# B&R Automation Studio project ABC_Pltzr (part 2)

### bgringbuffer.c
```c
#ifndef _BG_RINGBUFFER_C
#define _BG_RINGBUFFER_C
/*
File:
bgRingBuffer.c

About:
------
- ring buffer implementation

B&R System Dependencies:
------------------------
- B&R system library: none
- B&R system header files: stdarg.h

History:
--------
03/11/2005
-first version

Test and example code:
----------------------
- to run this file standalone:
--- enable following code section (remove or comment out #if 0 / #endif)
--- create cyclic object (task) from C Language and add this file
*/
#include <stdarg.h>

#include <bur/plctypes.h>
#ifdef _DEFAULT_INCLUDES
	#include <AsDefault.h>
#endif

#include "bgringbuffer.h"
//#include "bgdebug.h"

//#include "bgsprintf.h"
//#include "bgsprintf.c"

#if 0
#include<bur/plc.h>
#include <bur/plctypes.h>

//#include <bgsprintf.h>
#include <bgringbuffer.h>

_LOCAL int counter;

_LOCAL bgRingBuffer_typ myRB;

#define TXT_SIZE 64
_LOCAL char textBuffer1[TXT_SIZE];
_LOCAL char textBuffer2[TXT_SIZE];

#define RB_SIZE 64
_LOCAL char ringBuffer[RB_SIZE];

_INIT void Init(void) {

	rbInit(&myRB, ringBuffer, RB_SIZE);
}

_CYCLIC void Cyclic(void) {

	counter++;

	sprintf2(textBuffer1, "Counter=%d\n", counter);
	bgRingBuffPutString(&myRB, textBuffer1);
    bgRingBuffGet(&myRB, textBuffer2, TXT_SIZE);
}
#endif
/*End: Example/Test code*/

static char *bgRingBuffGetPtrToFileName(char *pFileNameWithPath)
{
/*
Input Example:
*pFileNameWithPath = "d:/data/temp/cobble/2005-9-1/new_ng.pgp/pgm/new_ng/cpu/bgstatemachine.c"
                                                                             |
Output value is ptr to: bgstatemachine.c ------------------------------------+
*/
int i;
int len = brsstrlen((UDINT)pFileNameWithPath);
char* pStart = (char*)(pFileNameWithPath + len);
	for(i=0;i<len; i++, pStart--){
		if( (*pStart == '/') || (*pStart == '\\') ){
			pStart++;
			return pStart;
		}
	}
	return pFileNameWithPath;
}

static void bgRingBuffIncDataInPtr(bgRingBuffer_typ *rb){
	rb->ptrDataIn++;
    if(rb->ptrDataIn >= rb->ptrCircularBufferEnd){
    	rb->ptrDataIn = rb->ptrCircularBufferBegin;
#if 0
/*mark wrap arround for testing*/
    	*rb->ptrDataIn = '@';
    	rb->ptrDataIn++;
#endif
    }
}

static void bgRingBuffIncDataOutPtr(bgRingBuffer_typ *rb){
	rb->ptrDataOut++;
	if(rb->ptrDataOut >= rb->ptrCircularBufferEnd)
		rb->ptrDataOut = rb->ptrCircularBufferBegin;
}

void bgRingBuffInit(bgRingBuffer_typ *rb, char *buffer, int bufSize)
{
	if(!buffer || !bufSize)
		return;

	rb->init = 1;
	rb->overrun = 0;
	rb->bufSize = bufSize;
    rb->ptrCircularBufferBegin = buffer;
    rb->ptrCircularBufferEnd = buffer + rb->bufSize;
    rb->ptrDataIn = rb->ptrCircularBufferBegin;
    rb->ptrDataOut = rb->ptrCircularBufferBegin;
}
/*
----------------------------------------------------------
*/
void bgRingBuffPutString(bgRingBuffer_typ *rb, char *sourceString)
{
    char *src = sourceString;

	if(!rb->init)
		return;

    /*input is string! look for zero termination*/
    while( *src ){

        /*store char*/
        *rb->ptrDataIn = *src;

        /*inc ptrs*/
		src++;

        bgRingBuffIncDataInPtr(rb);

        /*check if ring-buffer full*/
        if(rb->ptrDataIn == rb->ptrDataOut){
        	/*move out ptr one step ahead of in ptr*/
	        bgRingBuffIncDataOutPtr(rb);

			/*mark ring buffer overrun*/
			if(!rb->overrun){
		        char text[3]={'<','?','>'};
		        int i;
				rb->overrun = 1;
	        	for(i=0;i<3;i++){
			        *rb->ptrDataIn = text[i];
			        bgRingBuffIncDataInPtr(rb);
			        bgRingBuffIncDataOutPtr(rb);
		        }
		    }
        }
    }
}
/*
----------------------------------------------------------
*/
int bgRingBuffGet(bgRingBuffer_typ *rb, char *destination, int destSize)
{
char *dst = destination;
char *dstMax = dst + destSize;
int length = 0;

	if(!rb->init)
		return 0;

    if(rb->ptrDataIn == rb->ptrDataOut)
        return 0;

    while(1){
        *dst = *rb->ptrDataOut;
		length++;

        dst++;
        /*check if max size riched*/
        if(dst >= dstMax)
            break;

  		bgRingBuffIncDataOutPtr(rb);

        /*check if ring-buffer empty*/
        if(rb->ptrDataIn == rb->ptrDataOut){

        	/*mark end of ring buffer overrun*/
			if(rb->overrun){
		        char text[3]={'<','!','>'};
		        int i;

				rb->overrun = 0;
	        	for(i=0;i<3;i++){
			        *dst = text[i];
			        dst++;
			        length++;
			        if(dst >= dstMax)
			            break;
		        }
		    }

            break;
        }
    }
    return length;
}

void bgRingBuffPutDbgInfo(bgRingBuffer_typ *rb, char *file, char *function, unsigned int level, unsigned int unused, char *format, ...)
{
char txt[256];

va_list args;

	/*if dbg entry level > then currently set dbg level -> exit*/
	if( level > rb->dbgLevel )
		return;

	/*timestap needed? default=no*/
	if( rb->dbgFormat & BG_DEBUG_FORMAT_LEVEL){
		switch(level){
			case 0: bgRingBuffPutString(rb, "CRT|"); break;
			case 1: bgRingBuffPutString(rb, "ERR|"); break;
			case 2: bgRingBuffPutString(rb, "WAR|"); break;
			case 3: bgRingBuffPutString(rb, "INF|"); break;
			case 4: bgRingBuffPutString(rb, "DBG|"); break;
			default: bgRingBuffPutString(rb, "???|"); break;
		}
	}

	/*timestap needed? default=no*/
	if( rb->dbgFormat & BG_DEBUG_FORMAT_TIMESTAMP){
//		bgsprintf(txt, "%s|", "2005-10-01 12:32:44.123" );
//		bgRingBuffPutString(rb, txt);
	}

	/*filename needed? default=no*/
	if( rb->dbgFormat & BG_DEBUG_FORMAT_FILENAME){
//		bgsprintf(txt, "%s|", bgRingBuffGetPtrToFileName(file) );
//		bgRingBuffPutString(rb, txt);
	}

	/*function name needed? default=no*/
	if( rb->dbgFormat & BG_DEBUG_FORMAT_FUNCTION){
//		bgsprintf(txt, "%s()|", function);
//		bgRingBuffPutString(rb, txt);
	}

    va_start( args, format );

//	bgvsprintf(txt, format, args);
//	bgvsprintf(txt, format, args);

	bgRingBuffPutString(rb, txt);
}

#if 0
void bgRingBuffPrintf(bgRingBuffer_typ *rb, char *format, ...)
{
char txt[256];
va_list ap;
int num;

    va_start( ap, format );

//	bgvsprintf(txt, format, args);

	num = __ofmt(0, txt, 256, format, ap);

	va_end(ap);
//	return num;

	bgRingBuffPutString(rb, txt);
}
#endif

#endif
/*EOF*/
```

### bgsscanf.h
```c
/*
File:
bgsscanf.h

About:
------
- short and limited implementation of the sscanf() function

*/
#ifndef _BG_SSCANF_H
#define _BG_SSCANF_H

#include <stdarg.h>

/*
Public data types:
-----------------
*/

/*
Public functions:
-----------------
*/
int bgsscanf(const char *out, const char *format, ...);

int bgvsscanf(const char *out, const char *format, va_list args);

#endif
```

### bgstring.c
```c
#ifndef _BG_STRING_C
#define _BG_STRING_C

#ifdef WIN32
#include "string.h"
#else
#include <bur/plctypes.h>
#endif
#include "bgstring.h"

/*
File:
bgString.c

About:
------
- implements  additional string manipulation functions

B&R System Dependencies:
------------------------
- B&R system library: libasstring.a
- B&R system header files: asstring.h

History:
--------
09/11/2005
- rectified issue with bgStringListLines() to properly handle zero length
input string

05/08/2005
-first version

Test and example code:
----------------------
- to run this file standalone:
--- enable following code section (remove or comment out #if 0 / #endif)
--- create cyclic object (task) from C Language and add this file
*/

#if 0
#include <bur/plc.h>
#include <bur/plctypes.h>

#define TXT_SIZE 64
_LOCAL char textBuffer1[TXT_SIZE];
_LOCAL char textBuffer2[TXT_SIZE];
_LOCAL int idxResult;
_LOCAL int idxStart;
_LOCAL int idxEnd;

_INIT void Init(void) {

	/*use defaults*/
	idxStart 	= -1;
	idxEnd 		= -1;
	/*start with empty strings*/
	textBuffer1[0] = 0;
	textBuffer2[0] = 0;
}

_CYCLIC void Cyclic(void) {

	idxResult = bgStrFind(textBuffer1, textBuffer2, start, end);

}
#endif

/*End: Example/Test code*/
int bgStrFind(char *s, char *sub, int idxStart, int idxEnd)
{
	int i, j;
	int subLen;
	char *ptrStr;
	char *ptrSub;

	/*exit if null ptrs*/
	if(!s || !sub)
		return -1;

	/*exit if zero strings*/
	if( !(*s) || !(*sub) )
		return -1;

	subLen = brsstrlen((UDINT)sub);

	/*check starting index: default = -1 -> start @ s[0]*/
	if(idxStart < 0)
		idxStart = 0;

	/*check end index: default = -1 -> end is sLength - subLength*/
	if(idxEnd < 0){
		idxEnd = brsstrlen((UDINT)s) - subLen;
	}

	/*check if start is beyond the end*/
	if(idxStart > idxEnd)
		return -1;

	/*search for string <sub> within the string <s>*/
	for(i=idxStart; i<=idxEnd; i++)
	{
		ptrStr = s + i;
		ptrSub = sub;

		for(j=0; j<subLen; j++, ptrStr++, ptrSub++)
		{
			if( *ptrStr!= *ptrSub)
				break;
		}

		if( j == subLen)
			return i;
	}

	return -1;
}

/*
bgStrFindEx - has an extra option
option = 0; same as bgStrFind
option = 1; before comparing, both strings are converted to lower case
*/
int bgStrFindEx(char *s, char *sub, int idxStart, int idxEnd, int option)
{
	int i, j;
	int subLen;
	char *ptrStr;
	char *ptrSub;

	/*exit if null ptrs*/
	if(!s || !sub)
		return -1;

	/*exit if zero strings*/
	if( !(*s) || !(*sub) )
		return -1;

	subLen = brsstrlen((UDINT)sub);

	/*check starting index: default = -1 -> start @ s[0]*/
	if(idxStart < 0)
		idxStart = 0;

	/*check end index: default = -1 -> end is sLength - subLength*/
	if(idxEnd < 0){
		idxEnd = brsstrlen((UDINT)s) - subLen;
	}

	/*check if start is beyond the end*/
	if(idxStart > idxEnd)
		return -1;

	/*search for string <sub> within the string <s>*/
	for(i=idxStart; i<=idxEnd; i++)
	{
		ptrStr = s + i;
		ptrSub = sub;

		for(j=0; j<subLen; j++, ptrStr++, ptrSub++)
		{
			if(!option){
				if( *ptrStr!= *ptrSub)
					break;
			}else{
				if( bgCharToLowerCase(*ptrStr) != bgCharToLowerCase(*ptrSub) )
					break;
			}
		}

		if( j == subLen)
			return i;
	}

	return -1;
}

int bgStrCpyN(char *dest, char *src, int maxNoOfCharsToCopy)
{
int i;

	/*maxNoOfCharsToCopy-1 - takes into consideration that supplied max
	length is usually the buffer size, 1 char is needed for null termination
	*/
	for(i=0; i<(maxNoOfCharsToCopy-1);i++){
		*(dest+i)=*(src+i);
		if(! (*(src+i) ) )
			break;
	}

	/*if max reached, terminate dest string*/
	if(i >= (maxNoOfCharsToCopy-1))
		*(dest+i)=0;

	/*string termination is not included in the string length*/
	return i;
}

int bgStrTrimCRLF(char *s)
{
int i;
char c;

	for(i=0;i<255;i++){

		c = s[i];

		if( !c )
			break;

		if( (c == 0xa) || (c == 0xd) ){
			s[i] = 0;
			break;
		}
	}

	return i;
}

int bgStrCpyNTrimLeadingSpaces(char *dest, char *src, int maxNoOfCharsToCopy)
{
int i;
int found;
char *srcStart;

	/*look for leading spaces*/
	found = 0;
	for(i=0; i<(maxNoOfCharsToCopy-1);i++){
		if( *(src+i) != ' ' ){
			srcStart = src + i;
			found = 1;
			break;
		}
	}

	if(!found){
	/*src string is all spaces->set destination to empty string*/
		*dest = 0;
		return 0;
	}

	return bgStrCpyN(dest, srcStart, maxNoOfCharsToCopy);
}

/*
copy string, don't go over the size of dest buffer, trim leading / trailing spaces / convert
to lower case
*/
int bgStrCpyNTrimSpcsToLwr(char *dest, char *src, int maxNoOfCharsToCopy)
{
int i;
char* srcStart = src;
char* srcEnd;
int len = brsstrlen((UDINT)src);

	if( !len )
		return len;

	/*find src start, avoid leading spaces*/
	while(1){
		if( *srcStart != ' ')
			break;

		if( *srcStart == 0)
			return 0;

		srcStart++;
	}

	/*find src end, trim trailing spaces*/
	srcEnd = (char*)(src + len - 1);
	while(1){
		if( *srcEnd != ' ')
			break;

		if( *srcEnd == 0)
			return 0;

		srcEnd--;
	}

	srcEnd++;

	if( srcStart >= srcEnd )
		return 0;

	for(i=0; i<(maxNoOfCharsToCopy-1); i++){
		dest[i] = bgCharToLowerCase(*srcStart);
		srcStart++;
		if(srcStart >= srcEnd){
			i++;
			break;
		}
	}

	dest[i] = 0;
	return i;
}

int bgIsDigit(char c){
	return ((c>='0') && (c<='9')) ? 1 : 0;
}

#if 0
/*
Test for: bgStringListLinesEx()

The xxxxEx functions use externaly supplied buffer space to store result pointers to
lines / words.
Based on the supplied buffer size, functions will calculate max. number of items (char ptr-s)
that may be stored within the given / allocated storage area.
See: pList->itemCountMax

To test it out, create a new cyclic task then use following code!
*/
#include <bur/plc.h>
#include <bur/plctypes.h>

#include "bglib/bgString.h"
#include "bglib/bgString.c"

#include "bglib/bgdebug.h"
#include "bglib/bgringbuffer.c"

_LOCAL bgStringListEx_typ listLines;
_LOCAL bgStringListEx_typ listWords;
_LOCAL char multiLineTextBuffer[256];
_LOCAL int lineCount;
_LOCAL int wordCount;
_LOCAL int test;
_LOCAL char listPtrBuf[128];    /*this is a "free" storage for list ptr-s! use it with caution!*/

_INIT void init()
{
	strcpy(multiLineTextBuffer, "hello world\r\nThis is a test for second line!\r\nThird line is here and there...\r\nLine #4 : right.left dot !\r\n");
	test = 0;
}

_CYCLIC void cyclic()
{
int i, j;

/*
This is just an example on how to use external / user supplied buffer in order to
store line / word lists. Based on the supplied buffer size, functions will calculate
max. number of items that may be stored within the given / allocated storage area.
See: pList->itemCountMax
*/
char* lineListStorage = &listPtrBuf[0];
char* wordListStorage = &listPtrBuf[64];

	if( test ){
		test = 0;

		lineCount = bgStringListLinesEx(&listLines, multiLineTextBuffer, lineListStorage, 64);
		DBG("multiLineTextBuffer has lineCount=%d lines. (same as listLines.itemCount= %d). Lines are:\r\n", lineCount, listLines.itemCount);
		for(i=0; i<listLines.itemCount; i++){
			DBG("Line[%d]->%s\r\n", i, listLines.items[i]);
			wordCount = bgStringSplitLineEx(&listWords, ' ', listLines.items[i], wordListStorage, 64);
				DBG("     Line[%d] has wordCount=%d words. (same as listWords.itemCount= %d). Words are:\r\n", i, wordCount, listWords.itemCount)
			for(j = 0; j<listWords.itemCount; j++)
				DBG("     Word[%d]->%s\r\n", j, listWords.items[j]);
		}
	}
}
#endif
int bgStringListLines(bgStringList_typ * p){
unsigned char *ptrItemStart, *ptrItemEnd;
int	calcItemCount;

/*
	length = strlen( p->src );
*/
	p->itemCount = 0;

	ptrItemStart = p->src;
	ptrItemEnd = p->src;

	if( *ptrItemStart == 0){
		return 0;
	}

/*process the rest; build list of item pointers*/
	calcItemCount 	= 0;
	while( 1 ){
		if( (*ptrItemEnd == 0x0D) || (*ptrItemEnd == 0x0A)){
			*ptrItemEnd = 0;
			p->items[calcItemCount] = ptrItemStart;
			ptrItemEnd++;

			/*check for an additional \r or \n*/
			if( (*ptrItemEnd == 0x0D) || (*ptrItemEnd == 0x0A)){
				ptrItemEnd++;
			}

			ptrItemStart = ptrItemEnd;
			calcItemCount++;

			if(calcItemCount >= BG_STRINGLIST_MAXITEMCOUNT){
				p->itemCount = calcItemCount;
				return -1;
			}

			/*check for an end of the src string*/
			if( (*ptrItemEnd == 0) ){
				p->itemCount = calcItemCount;
				return calcItemCount;
			}
		}else
		if( *ptrItemEnd == 0){
			p->items[calcItemCount] = ptrItemStart;
			calcItemCount++;
			break;
		}else
			ptrItemEnd++;
	}/*while*/

	p->itemCount = calcItemCount;
	return calcItemCount;
}

void bgStringListExMemSet(bgStringListEx_typ *p, char* pAddrListBuffer, int sizeListBuffer)
{
	/*NOTE: we are going to use supplied char buffer as the storage for the array of char ptr-s!*/
    p->items = (unsigned char**)pAddrListBuffer;

	p->itemCountMax = sizeListBuffer / sizeof(char*);
}

int bgStringListLinesEx(bgStringListEx_typ * p, char* pContentBuffer, char* pAddrListBuffer, int sizeListBuffer){
unsigned char *ptrItemStart, *ptrItemEnd;
int	calcItemCount;

    p->src = (unsigned char*)pContentBuffer;

    /*if mem data is defined, use it; otherwise, mem shall have been set using a separate call to xxxExMemSet()*/
    if(pAddrListBuffer && sizeListBuffer)
        bgStringListExMemSet(p, pAddrListBuffer, sizeListBuffer);

	p->itemCount = 0;

	ptrItemStart = p->src;
	ptrItemEnd = p->src;

	if( *ptrItemStart == 0){
		return 0;
	}

/*process the rest; build list of item pointers*/
	calcItemCount 	= 0;
	while( 1 ){
		if( (*ptrItemEnd == 0x0D) || (*ptrItemEnd == 0x0A)){
			*ptrItemEnd = 0;
			p->items[calcItemCount] = ptrItemStart;
			ptrItemEnd++;

			/*check for an additional \r or \n*/
			if( (*ptrItemEnd == 0x0D) || (*ptrItemEnd == 0x0A)){
				ptrItemEnd++;
			}

			ptrItemStart = ptrItemEnd;
			calcItemCount++;

			if(calcItemCount >= p->itemCountMax){
				p->itemCount = calcItemCount;
				return -1;
			}

			/*check for an end of the src string*/
			if( (*ptrItemEnd == 0) ){
				p->itemCount = calcItemCount;
				return calcItemCount;
			}
		}else
		if( *ptrItemEnd == 0){
			p->items[calcItemCount] = ptrItemStart;
			calcItemCount++;
			break;
		}else
			ptrItemEnd++;
	}/*while*/

	p->itemCount = calcItemCount;
	return calcItemCount;
}

#if 0
Example:
(AS: Make a "C" task; add <filename>.c to the task; copy & paste this code)
#######
#include <bur/plc.h>
#include <bur/plctypes.h>

#include "bgString.h"
#include "bgString.c"

#include "bgdebug.h"

_LOCAL bgStringList_typ myList;
_LOCAL bgStringList_typ mySplitList;
_LOCAL char buffer[256];
_LOCAL int lineCount;
_LOCAL int test;

_INIT void init()
{
	strcpy(buffer, "hello world\r\nwhat is new?\r\nthird line\r\nline #4\r\n");
	test = 0;
}

_CYCLIC void cyclic()
{
int i, j;

	if( test ){
		test = 0;
		myList.src = buffer;
		lineCount = bgStringListLines(&myList);

		for(i=0; i<myList.itemCount; i++){
			DBG("Line[%d]->%s\r\n", i, myList.items[i]);

			mySplitList.src = myList.items[i];
			lineCount = bgStringSplitLine(&mySplitList, ' ');
			for(j = 0; j<mySplitList.itemCount; j++)
				DBG("     Word[%d]->%s\r\n", j, mySplitList.items[j]);
		}
	}
}
######
The above code generates following output (debug telnet client):
>Line[0]->hello world
     Word[0]->hello
     Word[1]->world
Line[1]->what is new?
     Word[0]->what
     Word[1]->is
     Word[2]->new?
Line[2]->third line
     Word[0]->third
     Word[1]->line
Line[3]->line #4
     Word[0]->line
     Word[1]->#4

#endif
int bgStringSplitLine(bgStringList_typ * p, char separator){
unsigned char *ptrItemStart, *ptrItemEnd;
int	calcItemCount;

	p->itemCount = 0;

	ptrItemStart = p->src;
	ptrItemEnd = p->src;

/*process the rest; build list of item pointers*/
	calcItemCount 	= 0;
	while( 1 ){
		if( (*ptrItemEnd == separator) ){
			*ptrItemEnd = 0;
			p->items[calcItemCount] = ptrItemStart;
			ptrItemEnd++;

			calcItemCount++;

			/*check for an additional separtor */
			while( (*ptrItemEnd == separator) ){
				ptrItemEnd++;
				if( (*ptrItemEnd == 0) ){
					p->itemCount = calcItemCount;
					return calcItemCount;
				}
			}

			ptrItemStart = ptrItemEnd;

			if(calcItemCount >= BG_STRINGLIST_MAXITEMCOUNT){
				p->itemCount = calcItemCount;
				return -1;
			}

			/*check for an end of the src string*/
			if( (*ptrItemEnd == 0) ){
				p->itemCount = calcItemCount;
				return calcItemCount;
			}
		}else
		if( *ptrItemEnd == 0){
			p->items[calcItemCount] = ptrItemStart;
			calcItemCount++;
			break;
		}else
			ptrItemEnd++;
	}/*while*/

	p->itemCount = calcItemCount;
	return calcItemCount;
}

int bgStringSplitLineEx(bgStringListEx_typ * p, char separator, char* pLineBuffer, char* pAddrListBuffer, int sizeListBuffer){
unsigned char *ptrItemStart, *ptrItemEnd;
int	calcItemCount;

    p->src = (unsigned char*)pLineBuffer;

    /*if mem data is defined, use it; otherwise, mem shall have been set using a separate call to xxxExMemSet()*/
    if(pAddrListBuffer && sizeListBuffer)
        bgStringListExMemSet(p, pAddrListBuffer, sizeListBuffer);

	p->itemCount = 0;

	ptrItemStart = p->src;
	ptrItemEnd = p->src;

/*process the rest; build list of item pointers*/
	calcItemCount 	= 0;
	while( 1 ){
		if( (*ptrItemEnd == separator) ){
			*ptrItemEnd = 0;
			p->items[calcItemCount] = ptrItemStart;
			ptrItemEnd++;

			calcItemCount++;

			/*check for an additional separtor */
			while( (*ptrItemEnd == separator) ){
				ptrItemEnd++;
				if( (*ptrItemEnd == 0) ){
					p->itemCount = calcItemCount;
					return calcItemCount;
				}
			}

			ptrItemStart = ptrItemEnd;

			if(calcItemCount >= p->itemCountMax){
				p->itemCount = calcItemCount;
				return -1;
			}

			/*check for an end of the src string*/
			if( (*ptrItemEnd == 0) ){
				p->itemCount = calcItemCount;
				return calcItemCount;
			}
		}else
		if( *ptrItemEnd == 0){
			p->items[calcItemCount] = ptrItemStart;
			calcItemCount++;
			break;
		}else
			ptrItemEnd++;
	}/*while*/

	p->itemCount = calcItemCount;
	return calcItemCount;
}

char *bgStringLower(char *s)
{
int i;
char c;

	for(i=0;i<255;i++){

		c = s[i];

		if( !c )
			break;

		if( (c >= 'A') && (c <= 'Z') ){
			s[i] = c - 'A' + 'a';
		}
	}

	return s;
}

char bgCharToLowerCase(char c)
{
char charLowerCase = c;

	if( (c >= 'A') && (c <= 'Z') ){
		charLowerCase = c - 'A' + 'a';
	}

	return charLowerCase;
}

char *bgStringUpper(char *s)
{
int i;
char c;

	for(i=0;i<255;i++){

		c = s[i];

		if( !c )
			break;

		if( (c >= 'a') && (c <= 'z') ){
			s[i] = c - 'a' + 'A';
		}
	}

	return s;
}

int bgStringIsMatch(char *s1, char *s2, int minChrCount)
{
	if( !brsstrcmp((UDINT)s1, (UDINT)s2) ){
		return 1;
	}else
		return 0;

}

int bgIsNumber_uint(char *s)
{
int i;
char c;

	/*limit execution to 255: don't want cycle time violation due to wrong ptr*/
	for(i=0;i<255;i++){

		c = s[i];

		/*end of valid input string?*/
		if( !c && i)
			return 1;

		/*zero input string?*/
		if( !c && !i)
			return 0;

		/*check if digit or space*/
		if( !bgIsDigit(c) && (c != ' '))
			return 0;
	}

	return 0;
}

int bgIsNumber_int(char *s)
{
int i;
char c;

	/*limit execution to 255: don't want cycle time violation due to wrong ptr*/
	for(i=0;i<255;i++){

		c = s[i];

		/*end of valid input string?*/
		if( !c && i)
			return 1;

		/*zero input string?*/
		if( !c && !i)
			return 0;

		/*check if digit or space*/
		if( !bgIsDigit(c) && (c != ' ') && (c != '-')  && (c != '+'))
			return 0;
	}

	return 0;
}

int bgAsciiToUint(char *src, unsigned int *dst)
{

unsigned int value;

	if( !bgIsNumber_uint(src) )
		return 0;

#ifdef WIN32
	/*TODO!!!*/
	value = 0;
#else
	value = brsatoi((UDINT)src);
#endif

	*dst = value;

	return 1;
}

int bgAsciiToInt(char *src, unsigned int *dst)
{

unsigned int value;

	if( !bgIsNumber_int(src) )
		return 0;

#ifdef WIN32
	/*TODO!!!*/
	value = 0;
#else
	value = brsatoi((UDINT)src);
#endif
	*dst = value;

	return 1;
}

int bgStrCopyFromTo(char* src, int srcStartPosition, int srcEndPosition, char* dest)
{
/*
-copy part of the memory from the section of src (from srcStartPosition to srcEndPosition) to dest
-srcEndPosition is not included in the copy (last copied byte position is srcEndPosition-1)
-length of the copied string is (srcEndPosition - srcStartPosition)
Example:
src="01234567890"
srcStartPosition=3
srcEndPosition=7

dest="3456"

return value: number of bytes copied (i.e. length of the dest string)
*/
int size = 0;
int i;

	if( srcEndPosition >= srcStartPosition )
		size = srcEndPosition - srcStartPosition;

	/*do memcopy! end position char is not included in the copy!*/
	for(i=0; i<size; i++)
		dest[i] = src[srcStartPosition + i];

	/*terminate string*/
	dest[size] = 0;

	return size;
}

int bgStrFindEOL(char* src, int startPosition)
{
/*
- search supplied c string "src" (zero terminated!!!) for the eof
- start search at startPosition and look for the first '\n'
- return:
-1 		- EOF (\n) not found
>=0		- EOF position
*/
int position = startPosition;
int i = 0;

	while(1){
		/*end of line?*/
		if( src[position] == '\n' ){
			/*if \r preceeds \n, dec EOL position by 1*/
			if( position && (src[position-1] == '\r') )
				position--;

		 	return position;
		}

 		/*end of string?*/
		if( src[position] == 0 ) return -1;

		/*prevent endless loop*/
		if( ++i >= 4096 ) return -1;

		position++;
	}

	return -1;
}

#endif
/*EOF*/
```

### bgstringTest.c
```c
#include <bur/plc.h>
#include <bur/plctypes.h>

#include "bgString.h"
#include "bgString.c"

#include "bgdebug.h"

_LOCAL bgStringList_typ myList;
_LOCAL bgStringList_typ mySplitList;
_LOCAL char buffer[256];
_LOCAL int lineCount;
_LOCAL int testListLines;
_LOCAL int testUpper;
_LOCAL int testLower;

_INIT void init()
{
	brsstrcpy((UDINT)buffer, (UDINT)"hello world\r\nwhat is new?\r\nthird line\r\nline #4\r\n");
	testListLines = 0;
	testUpper = 0;
	testLower = 0;
}

_CYCLIC void cyclic()
{
int i, j;

	if( testListLines ){
		testListLines = 0;
		myList.src = buffer;
		lineCount = bgStringListLines(&myList);

		for(i=0; i<myList.itemCount; i++){
			DBG("Line[%d]->%s\r\n", i, myList.items[i]);

			mySplitList.src = myList.items[i];
			lineCount = bgStringSplitLine(&mySplitList, ' ');
			for(j = 0; j<mySplitList.itemCount; j++)
				DBG("     Word[%d]->'%s'\r\n", j, mySplitList.items[j]);
		}
	}

	if( testLower ){
		testLower = 0;
		DBG("Input String        : '%s'\r\n", buffer);
		bgStringLower( buffer );
		DBG("Input String (Lower): '%s'\r\n", buffer);
	}

	if( testUpper ){
		testUpper = 0;
		DBG("Input String        : '%s'\r\n", buffer);
		bgStringUpper( buffer );
		DBG("Input String (Upper): '%s'\r\n", buffer);
	}

}
```

### bgTcpSocketServer.c
```c
/*
File: bgTcpSocketServer.c
=====

B&R Libraries:
==============
Make sure to add following .a files to the task using this source file:
libsys_lib.a
libbrsystem.a
libastcp.a
*/

/*
B&R components:
===============================================================================
*/
#include <bur/plc.h>
#include <bur/plctypes.h>
#include <astcp.h>
#include <brsystem.h>
#include <sys_lib.h>

/*
BG components
===============================================================================
*/
#include "bgdebug.h"
#include "bgstring.h"
#include "bgsscanf.h"
#include "bgTcpSocketClientServer.h"

static void bgTcpSocketServerMemAlloc(bgTcpSocketServer_typ* p);
static void bgTcpSocketServerSessionStart(bgTcpSocketServer_typ* p);
static void bgTcpSocketServerSessionCyclic(bgTcpSocketServer_typ* p);
static void bgTcpSocketServerSessionStateMachine(bgTcpSocketSession_typ* pSession);
static void	bgTcpSocketServerExecuteSessionHandler(bgTcpSocketSession_typ* pSession, int init);
static void bgTcpSocketServerSessionSendData(bgTcpSocketSession_typ* pSession);
static void bgTcpSocketServerDefaultSessionHandler(bgTcpSocketSession_typ* pSession);
static void bgTcpSocketSendErrorResponse(bgTcpSocketSession_typ* pSession, int responseCode, char* msg);

/*
TCP Socket Server
######################################################################################################
######################################################################################################
######################################################################################################
######################################################################################################
*/
void bgTcpSocketServerInit(bgTcpSocketServer_typ* pServer,
    int portNumber,
    int numberOfSessions,
    int sessionSendBufSize,
    int sessionRecvBufSize,
    int applicationBufSize,
    void (*pSessionHandler)(bgTcpSocketSession_typ*),
    void (*pApplicationHandler)(bgTcpSocketSession_typ*))
{
    pServer->serverPort = portNumber;

    if(numberOfSessions <= BGTCPSOCKSRV_MAX_SESSIONS )
        pServer->numSupportedSessions = numberOfSessions;
    else{
        DBGCRT("bgTcpSocketServerInit(): max sessions= %d; %d sessions is to many!\r\n",
            BGTCPSOCKSRV_MAX_SESSIONS, numberOfSessions);
        pServer->numSupportedSessions = BGTCPSOCKSRV_MAX_SESSIONS;
    }

    pServer->sessionSendBufSize = sessionSendBufSize;

    pServer->sessionRecvBufSize = sessionRecvBufSize;

	pServer->applicationBufSize = applicationBufSize;

    pServer->sessionTotalBufSize = pServer->sessionSendBufSize + pServer->sessionRecvBufSize + pServer->applicationBufSize;

    pServer->totalBufSize = pServer->sessionTotalBufSize * pServer->numSupportedSessions;

    pServer->pSessionHandler = pSessionHandler;

    pServer->pApplicationHandler = pApplicationHandler;

	pServer->sockStateData = BGTCPSOCK_STATE_INITOPEN;

	pServer->dbgDumpSendBuf = 0;
	pServer->dbgDumpRecvBuf = 0;

	/*allocate memory for send/recv buffers*/
	bgTcpSocketServerMemAlloc(pServer);

	if(pServer->memAllocStatus2){
			DBGCRT("bgTcpSocketServerCyclic: memory alloc error! memAllocStatus2=%d\r\n", pServer->memAllocStatus2);
	}
}

void bgTcpSocketServerCyclic(bgTcpSocketServer_typ* pServer)
{
int i;

	/*if memalloc fails, can't do much!*/
	if(pServer->memAllocStatus2)
		return;

	/*execute session state machine*/
	bgTcpSocketServerSessionCyclic(pServer);

	/*server state machine*/
	switch(pServer->sockStateData){
		case BGTCPSOCK_STATE_NONE:
    		return;
		break;

		case BGTCPSOCK_STATE_INITOPEN:
			pServer->tcpOpen.enable = 1;
			pServer->tcpOpen.port = pServer->serverPort;        /* server listening port number*/
			pServer->tcpOpen.pIfAddr = 0;
			pServer->tcpOpen.options = tcpOPT_REUSEADDR;
    		pServer->sockStateData = BGTCPSOCK_STATE_OPEN;
		break;

        case BGTCPSOCK_STATE_OPEN:
			TcpOpen(&pServer->tcpOpen);

			if( pServer->tcpOpen.status == 0xFFFF )
				return;

			if( !pServer->tcpOpen.status ){
				pServer->tcpServer.enable = 1;
				pServer->tcpServer.ident = pServer->tcpOpen.ident;
				pServer->tcpServer.backlog = 5;
	    		pServer->tcpServer.pIpAddr = (unsigned long)pServer->clientIpAddr;
				pServer->sockStateData = BGTCPSOCK_STATE_LISTEN;

                /*clear all sessions*/
                for(i=0; i < BGTCPSOCKSRV_MAX_SESSIONS; i++){
                    pServer->session[i].ident = i;
                    pServer->session[i].socketState = BGTCPSOCK_SESSION_STATE_NONE;
                }

				return;
			}

            /* TODO: TcpOpen error handling! */
			pServer->sockStateData = BGTCPSOCK_STATE_NONE;
		break;

        case BGTCPSOCK_STATE_LISTEN:
    		TcpServer(&pServer->tcpServer);					/* wait connections from the clients */

			if(pServer->tcpServer.status == 0xFFFF)
				return;

			if(!pServer->tcpServer.status){
                bgTcpSocketServerSessionStart(pServer);
				return;
			}

            /*TODO: what to do on error?*/
			goto errorExit;
		break;

        case BGTCPSOCK_STATE_TOOBUSY:
            if( pServer->numActiveSessions < pServer->numSupportedSessions ){
                DBGMSG("bgTcpSocketServerCyclic(): session available, restaring server listening\r\n");
    			pServer->sockStateData = BGTCPSOCK_STATE_LISTEN;
            }

            /*TODO: implement timeout here -> kill sessions if stuck*/
        break;
	 }

    return;

errorExit:

/*TODO: what to do on error?*/
	DBGCRT("bgTcpSocketServer: ERROR! tcpServer.status=%d\r\n", pServer->tcpServer.status);
	return;
}

static void bgTcpSocketServerMemAlloc(bgTcpSocketServer_typ* pServer)
{
unsigned int memSize;
int i;

	/*Get System Memory Information*/
	pServer->MEMInfo.enable = 1;
	MEMInfo(&pServer->MEMInfo);

	memSize = pServer->totalBufSize;

	/*allocate space for send/recv buffers*/
	if(pServer->sendRecvBuffer == 0){
		/* allocate new memory from RAM*/
    	pServer->memAllocStatus2 = TMP_alloc(memSize, (void**)&pServer->sendRecvBuffer);
	}else{
		/*memory is allready allocated -> free it first!*/
    	pServer->memAllocStatus2 = TMP_free(memSize, (void**)pServer->sendRecvBuffer);

    	/*allocate new memory from RAM*/
    	pServer->memAllocStatus2 = TMP_alloc(memSize, (void**)pServer->sendRecvBuffer);
	}

	/*assign send/recv buffer ptrs*/
    for(i=0; i < pServer->numSupportedSessions; i++){
        pServer->session[i].pSendBuf = (char*)(pServer->sendRecvBuffer + i * pServer->sessionTotalBufSize);
		pServer->session[i].sendBufLength = pServer->sessionSendBufSize;

        pServer->session[i].pRecvBuf = (char*)(pServer->session[i].pSendBuf + pServer->sessionSendBufSize);
		pServer->session[i].recvBufLength = pServer->sessionRecvBufSize;

        pServer->session[i].pAppBuf = (char*)(pServer->session[i].pRecvBuf + pServer->sessionRecvBufSize);
		pServer->session[i].appBufLength = pServer->applicationBufSize;
    }
}

static void bgTcpSocketServerSessionStart(bgTcpSocketServer_typ* pServer)
{
int i;
bgTcpSocketSession_typ *pSession;

    for(i=0; i < pServer->numSupportedSessions; i++){
        if( pServer->session[i].socketState == BGTCPSOCK_SESSION_STATE_NONE){
            pSession = &pServer->session[i];
            pSession->socketState = BGTCPSOCK_SESSION_STATE_RECEIVE;

			pSession->tcpSend.enable = 1;
			pSession->tcpSend.ident = pServer->tcpServer.identclnt;   /* copy the  Ident number */
			pSession->tcpSend.flags = 0;
			pSession->tcpSend.pData = (UDINT)pSession->pSendBuf;

			pSession->tcpRecv.enable = 1;
			pSession->tcpRecv.ident = pServer->tcpServer.identclnt;     /* copy the  Ident number */
			pSession->tcpRecv.pData = (UDINT)pSession->pRecvBuf;        /* address of the buffer */;
			pSession->tcpRecv.datamax = pSession->recvBufLength;    	/* length of the buffer */;

			pSession->tcpClose.enable = 1;
   			pSession->tcpClose.ident = pServer->tcpServer.identclnt;    /* copy the  Ident number */

			pSession->pTcpLayer = (char*)pServer;	                    /*each session has ptr to tcp layer (client or server) data*/

            pSession->rxByteCountTotal = 0;
            pSession->txByteCountTotal = 0;
            pSession->rxByteCount = 0;
            pSession->txByteCount = 0;
            brsstrcpy((UDINT)pSession->clientIpAddr, (UDINT)pServer->clientIpAddr);

			pSession->dbgDumpRecvBuf = pServer->dbgDumpRecvBuf;
			pSession->dbgDumpSendBuf = pServer->dbgDumpSendBuf;

			/*init session specific handler - call the handler with init pSession->flag=1*/
			bgTcpSocketServerExecuteSessionHandler(pSession, 1);

			DBGMSG("bgTcpSocketServerSessionStart(): connection from %s, starting session Id= %d\r\n", pServer->clientIpAddr, i);
            return;
        }
    }

	DBGCRT("bgTcpSocketServerSessionStart(): server busy! activeSessions= %d\r\n", pServer->numSupportedSessions);
    pServer->sockStateData = BGTCPSOCK_STATE_TOOBUSY;
}

static void bgTcpSocketServerSessionCyclic(bgTcpSocketServer_typ* pServer)
{
int i;
bgTcpSocketSession_typ *pSession;
int activeSessions = 0;

    for(i=0; i < pServer->numSupportedSessions; i++){
        pSession = &pServer->session[i];

        if( pSession->socketState != BGTCPSOCK_SESSION_STATE_NONE){
            activeSessions++;
            bgTcpSocketServerSessionStateMachine(pSession);
        }
    }
    pServer->numActiveSessions = activeSessions;
}

static void bgTcpSocketServerSessionStateMachine(bgTcpSocketSession_typ* pSession)
{
    switch(pSession->socketState){
		case BGTCPSOCK_SESSION_STATE_SEND:

            TcpSend(&pSession->tcpSend);            				/* send the data */

            if(!pSession->tcpSend.status){
            	pSession->txByteCount += pSession->tcpSend.sentlen;

				DBGMSG("bgTcpSocketServerSessionStateMachine(): SEND complete! status=%d; curLen=%d; cumLen=%d\r\n",
					pSession->tcpSend.status, pSession->tcpSend.sentlen,
					pSession->txByteCount);
/*
following simplifies testing of multiple sessions:
for normal operation use
#if 1
for delayed operation (testing) use
#if 0
*/
#if 1
    			pSession->socketState = BGTCPSOCK_SESSION_STATE_CLOSE;
#else
    			p->socketState = BGTCPSOCK_SESSION_STATE_DELAY;
				p->delayCounter = 50;
#endif
				break;
			}

			/*in case of the following error -> close connection*/
            if( (pSession->tcpSend.status == 27210) 	||
            	(pSession->tcpSend.status == 27135)	||
            	(pSession->tcpSend.status == tcpERR_NOT_CONNECTED)	||
            	(pSession->tcpSend.status == tcpERR_SYSTEM)	||
            	(pSession->tcpSend.status == 27249)
            ){
				DBGMSG("bgTcpSocketServerSessionStateMachine(): SEND error=%d\r\n", pSession->tcpSend.status);
    			pSession->socketState = BGTCPSOCK_SESSION_STATE_CLOSE;
				break;
			}else
			if(pSession->tcpSend.status == tcpERR_SENTLEN){
				/*long send! call send buf handler to fill in more data*/
			    if(pSession->pSendBufHandler){
    				(*pSession->pSendBufHandler)(pSession);

					DBGMSG("bgHttpSendBufCallback(): SEND status=%d; curLen=%d; cumLen=%d; remLen=%d\r\n",
						pSession->tcpSend.status,
						pSession->tcpSend.sentlen,
						pSession->txByteCount,
						pSession->tcpSend.datalen);
			    }
				else{
					DBGMSG("bgTcpSocketServerSessionStateMachine(): SEND incomplete! sendBuf handler NOT defined!? status=%d\r\n", pSession->tcpSend.status);
		   			pSession->socketState = BGTCPSOCK_SESSION_STATE_CLOSE;
				}
			}else{
				DBGMSG("bgTcpSocketServerSessionStateMachine(): SEND status=%d\r\n", pSession->tcpSend.status);
 			}

		break;

		case BGTCPSOCK_SESSION_STATE_RECEIVE:
            TcpRecv(&pSession->tcpRecv);          				/* recv data*/

            if(!pSession->tcpRecv.status){
                if(pSession->tcpRecv.recvlen){
					bgTcpSocketServerExecuteSessionHandler(pSession, 0);
                }else{
					/*remote socket has closed*/
    				pSession->socketState = BGTCPSOCK_SESSION_STATE_CLOSE;    /*close this server socket*/
				}
            }
		break;

		case BGTCPSOCK_SESSION_STATE_CLOSE:
			pSession->tcpClose.how = tcpSHUT_RD & tcpSHUT_WR;

            TcpClose(&pSession->tcpClose);          				/* set the socket free */

			if(pSession->tcpClose.status == 0xFFFF)
				return;

	    	pSession->socketState = BGTCPSOCK_SESSION_STATE_NONE;
			DBGMSG("bgTcpSocketServerSessionStateMachine(): stopping session Id= %d\r\n", pSession->ident);
		break;

		case BGTCPSOCK_SESSION_STATE_DELAY:
			pSession->delayCounter--;
			if(pSession->delayCounter <= 0)
    			pSession->socketState = BGTCPSOCK_SESSION_STATE_CLOSE;    /*close this server socket*/
		break;

		default:

		break;
	}
}

static void	bgTcpSocketServerExecuteSessionHandler(bgTcpSocketSession_typ* pSession, int init)
{
bgTcpSocketServer_typ* pServer = (bgTcpSocketServer_typ*)pSession->pTcpLayer;

	pSession->init = 0;
	if( init )
		pSession->init = 1;

    if(pServer->pSessionHandler)
    	(*pServer->pSessionHandler)(pSession);
    else
    	bgTcpSocketServerDefaultSessionHandler(pSession);

	pSession->init = 0;

	/*has upper layer requested action!?*/
	if( pSession->bSendData ){
		pSession->bSendData = 0;
		bgTcpSocketServerSessionSendData(pSession);
	}
}

static void bgTcpSocketServerSessionSendData(bgTcpSocketSession_typ* pSession)
{
	pSession->tcpSend.datalen = pSession->txByteCountTotal;
	pSession->socketState = BGTCPSOCK_SESSION_STATE_SEND;
}

/*
Default session handler
######################################################################################################
######################################################################################################
######################################################################################################
######################################################################################################
*/
static void bgTcpSocketServerDefaultSessionHandler(bgTcpSocketSession_typ* pSession)
{
    /*default session handler -> send out http error response "internal server error"*/
    bgTcpSocketSendErrorResponse(pSession, 500, "Internal server error. (Session handler not installed.)");
}

static void bgTcpSocketSendErrorResponse(bgTcpSocketSession_typ* pSession, int responseCode, char *msg)
{
char textBuffer[256];
char* pDst = pSession->pSendBuf;
int len;

	pDst[0]=0;
	bgsprintf(textBuffer, "%s %d %s\r\n", BGHTTP_CONST_STRING_VERSION, responseCode, msg );
	brsstrcpy((UDINT)pDst, (UDINT)textBuffer);

	len = brsstrlen((UDINT)pSession->pSendBuf);
	pSession->txByteCountTotal = len;
	bgTcpSocketServerSessionSendData(pSession);
}
```

### bgTimer1ms.h
```c
#ifndef _BG_TIMER1MS_H
#define _BG_TIMER1MS_H

#include <bur/plc.h>
#include <bur/plctypes.h>
#include <standard.h>

void bgTimerExecute(TON_typ *timer);
void bgTimerStart(TON_typ *timer, int timeoutTime);
void bgTimerStop(TON_typ *timer);
void bgTimerReset(TON_typ *timer);
int	bgTimerIsTimeOut(TON_typ *timer);
int	bgTimerTimeRemaining(TON_typ *timer);

#endif
```

### bgTimer.c
```c
#include "bgTimer.h"

void bgTimerExecute(TON_10ms_typ *timer){
	TON_10ms(timer);
}

void bgTimerStart(TON_10ms_typ *timer, int timeoutTime){
	timer->IN = 0;
	TON_10ms(timer);
	timer->IN = 1;
	timer->PT = timeoutTime;
	TON_10ms(timer );
}

void bgTimerStop(TON_10ms_typ *timer){
	timer->IN = 0;
	TON_10ms(timer);
}
int  bgTimerIsTimeOut(TON_10ms_typ *timer){
	return timer->Q;
}

int bgTimerTimeRemaining(TON_10ms_typ *timer){
	return (timer->PT - timer->ET);
}
```

### bgPVSerialize.c
```c
#ifndef _BG_SERIALIZE_C
#define _BG_SERIALIZE_C

#ifdef WIN32
#include "string.h"
#else
#include <bur/plctypes.h>
#include <sys_lib.h>
#endif

#include <AsBrStr.h>

//#include <string.h>
//#include <brsystem.h>
//#include <sys_lib.h>
//#include <asstring.h>
#include "bgstring.h"
//#include "bgsprintf.h"
#include "bgsscanf.h"
#include "bgsscanf.c"
#include "../Libraries/sprintf2/sprintf2.h"

#define PV_SERIALIZE_ITEM_DELIM_CRLF "\r\n"
#define PV_SERIALIZE_ITEM_DELIM_COMMA ","
//#define PV_SERIALIZE_STR_MARKUP "\""
#define PV_SERIALIZE_STR_MARKUP "'"

#define PV_SERIALIZE_ERR_ZEROPTR -1
#define PV_SERIALIZE_ERR_PVNOTFOUND -2
#define PV_SERIALIZE_ERR_PVADRNOTFOUND -3
#define PV_SERIALIZE_ERR_OBUFOVERFLOW -4
#define PV_SERIALIZE_ERR_NOCOMPARE -5 //comparison is not possible (i.e. different data structures)

#define PV_SERIALIZE_ERR_LAST -10

typedef struct bgPVSerialize_typ
{
	char* toOutStream;
	UDINT lengthOutStream;
	DINT outputCharCount;
	DINT errorCode;
	DINT arrayIndexFrom;
	DINT arrayIndexTo;
	char* pItemDelim;
	char* pStrMarkup;

}bgPVSerialize_typ;

static void bgPVSubStructSerialize(bgPVSerialize_typ* p, char* pvNameRoot, char* pvName, UINT dimension);
static void bgPVSerialize(bgPVSerialize_typ* p, char* pvNameRoot, char* pvName);
static void bgPVSubStructCompare(bgPVSerialize_typ* p, char* pvNameRoot, char* pvName, UINT dimension, char* pvNameRoot2);
static void bgPVCompare(bgPVSerialize_typ* p, char* pvNameRoot, char* pvName, char* pvNameRoot2);

//#ifndef DBG
//#define DBG() ;
//#endif

#define PV_TYPE_MAX_INDEX	24
#if 0
static const char *bgPVTypeStrings[PV_TYPE_MAX_INDEX + 1]={
	"STRUCT",	/*0*/
	"BOOL",		/*1*/
	"SINT",		/*2*/
	"INT",		/*3*/
	"DINT",		/*4*/
	"USINT",		/*5*/
	"UINT",		/*6*/
	"UDINT",		/*7*/
	"REAL",		/*8*/
	"STRING ",	/*9*/
	"ULINT",		/*10*/
	"DATETIME",	/*11*/
	"TIME",		/*12*/
	"DATE",		/*13*/
	"LREAL",		/*14*/
	"ARRAY",		/*15*/
	"TIME_OF_DAY",	/*16*/
	"BYTE",		/*17*/
	"WORD",		/*18*/
	"DWORD",	/*19*/
	"LWORD",	/*20*/
	"WSTRING",	/*21*/
	"?22",		/*22*/
	"LINT",		/*23*/
	};
static const char *bgGetPVTypeString(int pvTypeIndex){
	if(pvTypeIndex >= PV_TYPE_MAX_INDEX){
		return "TYPE=?";
	}

	return bgPVTypeStrings[pvTypeIndex];
}
#endif

static void bgGetPVValueText(char* pvValue, UDINT data_typ, UDINT data_len, UINT dimension, UDINT adr)
{
/*
	if( dimension != 1)
		DBG("TODO: display multidimensional values...");
*/
	switch(data_typ){
		case PB_DT_STRUCT:
			//DBG("TODO: display struct values...");
			break;
		case PB_DT_BOOL:
			sprintf2(pvValue, "%d", *( (char*)adr ));
			break;
		case PB_DT_INT8:
			sprintf2(pvValue, "%d", *( (char*)adr) );
			break;
		case PB_DT_INT16:
			sprintf2(pvValue, "%d", *( (short*)adr ) );
			break;
		case PB_DT_INT32:
			sprintf2(pvValue, "%d", *( (int*)adr ));
			break;
		case PB_DT_BYTE:
			sprintf2(pvValue, "%u", *( (unsigned char*)adr));
			break;
		case PB_DT_WORD:
			sprintf2(pvValue, "%u", *( (unsigned short*)adr));
			break;
		case PB_DT_LONG:
			sprintf2(pvValue, "%u", *( (unsigned int*)adr));
			break;
		case PB_DT_FLOAT:
			{
				char temp[32];
				brsftoa( *((float*)adr), (UDINT)temp);
				sprintf2(pvValue, "%s", temp);
			}
			break;
		case PB_DT_VIS:
			sprintf2(pvValue, "%s", (char*)adr );
			break;
		case PB_DT_OCTET:
			//DBG("TODO: display octet values...");
			break;
		case PB_DT_DATE:
			//DBG("TODO: display date values...");
			break;
		case PB_DT_TIME:
			//DBG("TODO: display time values...");
			break;
		case PB_DT_DIFF:
			//DBG("TODO: display time-diff values...");
			break;
		case 14://double
			{
				char temp[32];
				double value_double = *((double*)(adr));
				float value_float = (float)value_double;
				brsftoa( value_float, (UDINT)temp);
				sprintf2(pvValue, "%s", temp);
			}
			break;
		case PB_DT_ARRAY:
			//DBG("TODO: display array values...");
			break;
	}
}

static void bgSetPVValueText(char* pvValue, UDINT data_typ, UDINT data_len, UINT dimension, UDINT adr)
{
/*
	if( dimension != 1)
		DBG("TODO: display multidimensional values...");
*/
	switch(data_typ){
		case PB_DT_STRUCT:
			//DBG("TODO: set struct values...");
			break;
		case PB_DT_BOOL:
			bgsscanf(pvValue, "%d", (char*)adr );
			break;
		case PB_DT_INT8:
			bgsscanf(pvValue, "%d", (char*)adr );
			break;
		case PB_DT_INT16:
			bgsscanf(pvValue, "%d", (short*)adr  );
			break;
		case PB_DT_INT32:
			bgsscanf(pvValue, "%d", (int*)adr );
			break;
		case PB_DT_BYTE:
			bgsscanf(pvValue, "%u", (unsigned char*)adr);
			break;
		case PB_DT_WORD:
			bgsscanf(pvValue, "%u", (unsigned short*)adr);
			break;
		case PB_DT_LONG:
			bgsscanf(pvValue, "%u", (unsigned int*)adr);
			break;
		case PB_DT_FLOAT:
			{
				*((float*)adr) = brsatof((UDINT)pvValue);
			}
			break;
		case PB_DT_VIS:
			{
				int ii=0;
				//copy string
				//don't copy over the size of the dest buffer!
				//terminate properly
				char* src=(char*)pvValue;
				char* dst=(char*)adr;
				//DBG("GBTST= %s len=%d", src, data_len);
				for(ii=0; ii<data_len; ii++){
					dst[ii] = src[ii];
					//if end of src string > exit
					if(!src[ii])
						break;
				}
				//src longer than dst > terminate dst
				dst[data_len-1] = 0;
			}
			break;
		case PB_DT_OCTET:
			//DBG("TODO: display octet values...");
			break;
		case PB_DT_DATE:
			//DBG("TODO: display date values...");
			break;
		case PB_DT_TIME:
			//DBG("TODO: display time values...");
			break;
		case PB_DT_DIFF:
			//DBG("TODO: display time-diff values...");
			break;
		case 14://double
			{
				float value_float = brsatof((UDINT)pvValue);
				double value_double = (double)value_float;
				*((double*)adr) = value_double;
			}
			break;
		case PB_DT_ARRAY:
			//DBG("TODO: display array values...");
			break;
	}
}

static void bgPVWriteOutStream(bgPVSerialize_typ* p, char* pvName, char* pvTextValue)
{
	if(!p || !p->toOutStream || !pvName || !pvTextValue || !p->pItemDelim)
		return;

	brsstrcat((UDINT)p->toOutStream, (UDINT)pvName);
	brsstrcat((UDINT)p->toOutStream, (UDINT)"=");
	brsstrcat((UDINT)p->toOutStream, (UDINT)pvTextValue);
	brsstrcat((UDINT)p->toOutStream, (UDINT)p->pItemDelim);	// delimiter "\r\n" or ","

	p->outputCharCount += brsstrlen((UDINT)pvName);
	p->outputCharCount += brsstrlen((UDINT)pvTextValue);
	p->outputCharCount += brsstrlen((UDINT)p->pItemDelim) + 1; //  '=' + sizeof the delimiter string

	if(p->outputCharCount >= (p->lengthOutStream - 100) ){//TODO: needs to be a better way to handle output buffer overflow
		p->errorCode = PV_SERIALIZE_ERR_OBUFOVERFLOW;
		return;
	}
}

static void bgTxtWriteOutStream(bgPVSerialize_typ* p, char* pTxt)
{
	if(!p || !p->toOutStream || !pTxt)
		return;

	brsstrcat((UDINT)p->toOutStream, (UDINT)pTxt);

	p->outputCharCount += brsstrlen((UDINT)pTxt);

	if(p->outputCharCount >= (p->lengthOutStream - 100) ){//TODO: needs to be a better way to handle output buffer overflow
		p->errorCode = PV_SERIALIZE_ERR_OBUFOVERFLOW;
		return;
	}
}

static int bgPVSerializeIsArray(int data_typ, int data_len, int dimension)
{
	if(data_typ && (dimension > 1)){
		return 1;
	}
	return 0;
}

static void bgPVArraySerialize(bgPVSerialize_typ* p, char* pvNameRoot, char* pvName, int dimension)
{
	int ii = 0;
	// TODO: checking for max size of the strings that are copied to these arrays
	char structName[256];
	char structItemName[32];

	for(ii=0; ii < dimension; ii++){
		// NOTE: verify why PV_item destroys content of the buffer supplied as 1st param
		if( !pvName){
			brsstrcpy((UDINT)structName, (UDINT)pvNameRoot);
		}else{
			brsstrcpy((UDINT)structName, (UDINT)pvNameRoot);
			//strcat(structName, ".");
			//strcat(structName, pvName);
		}

		{
			char arrayIndexTxt[10];
			brsstrcpy((UDINT)structItemName, (UDINT)pvName);
			brsstrcat((UDINT)structItemName, (UDINT)"[");
			brsitoa(ii, (UDINT)arrayIndexTxt);
			brsstrcat((UDINT)structItemName, (UDINT)arrayIndexTxt);
			brsstrcat((UDINT)structItemName, (UDINT)"]");
		}

		bgPVSerialize(p, structName, structItemName);

		if(p->errorCode)
			return;

	}
}

static void bgPVArraySerializeRootToFrom(bgPVSerialize_typ* p, char* pvNameRoot, int dimension)
{
	int ii = 0;
	// TODO: checking for max size of the strings that are copied to these arrays
	char structItemName[32];

	for(ii = p->arrayIndexFrom; (ii < dimension) && (ii <= p->arrayIndexTo); ii++){
		// NOTE: verify why PV_item destroys content of the buffer supplied as 1st param
		{
			char arrayIndexTxt[10];
			brsstrcpy((UDINT)structItemName, (UDINT)pvNameRoot);
			brsstrcat((UDINT)structItemName, (UDINT)"[");
			brsitoa(ii, (UDINT)arrayIndexTxt);
			brsstrcat((UDINT)structItemName, (UDINT)arrayIndexTxt);
			brsstrcat((UDINT)structItemName, (UDINT)"]");
		}
		bgTxtWriteOutStream(p, structItemName);
		bgTxtWriteOutStream(p, "=[");
		bgPVSerialize(p, structItemName, 0);
		//bgTxtWriteOutStream(p, "]\r\n");
		bgTxtWriteOutStream(p, "],");

		if(p->errorCode)
			return;
	}
}

static void bgPVSerialize(bgPVSerialize_typ* p, char* pvNameRoot, char* pvName)
{
	UINT status;
	UDINT data_typ;
	UDINT data_len;
	UINT dimension;
	UDINT adr;
	char structItemPVName[256];

	if( !pvName){
		brsstrcpy((UDINT)structItemPVName, (UDINT)pvNameRoot);

	}else{
		brsstrcpy((UDINT)structItemPVName, (UDINT)pvNameRoot);
		brsstrcat((UDINT)structItemPVName, (UDINT)".");
		brsstrcat((UDINT)structItemPVName, (UDINT)pvName);
	}

	status = PV_ninfo(structItemPVName, &data_typ, &data_len, &dimension);

	if( status ){
		p->errorCode = status;
		return;
	}

	if( bgPVSerializeIsArray(data_typ, data_len, dimension) ){
		bgPVArraySerialize(p, pvNameRoot, pvName, dimension);
		return;
	}

	status = PV_xgetadr(structItemPVName, &adr, &data_len);

	if( status ){
		p->errorCode = status;
		return;
	}

	if(data_typ == PB_DT_STRUCT){
		//DBG("PV='%s' Typ=%s Len=%d Dim=%d" , pvnamecomplete, bgGetPVTypeString(data_typ), data_len, dimension);
		bgPVSubStructSerialize(p, pvNameRoot, pvName, dimension);
	}else{
		char pvTextValue[256];
		int len = 0;

		if(data_typ == PB_DT_VIS){//STRING VALUES ONLY > marked with a special markup at the begining and end
			brsstrcpy((UDINT)pvTextValue, (UDINT)p->pStrMarkup);//set string begining markup (i.e. "\"")
			len = brsstrlen((UDINT)pvTextValue);
		}

		bgGetPVValueText(&pvTextValue[len], data_typ, data_len, dimension, adr);

		if(data_typ == PB_DT_VIS){//STRING VALUES ONLY > marked with a special markup at the begining and end
			brsstrcat((UDINT)pvTextValue, (UDINT)p->pStrMarkup);//set string ending markup (i.e. "\"")
		}

		//DBG("stritemPV='%s' Typ=%s Len=%d Dim=%d Val=%s" , pvName, bgGetPVTypeString(data_typ), data_len, dimension, pvTextValue);
		bgPVWriteOutStream(p, pvName, pvTextValue);
	}

}

static void bgPVSubStructSerialize(bgPVSerialize_typ* p, char* pvNameRoot, char* pvName, UINT dimension)
{
/*
Example:
typedef struct str1_typ{
UINT val1;
UINT val2;
}str1_typ;

typedef struct str2_typ{
UINT val3;
}str2_typ;

typedef struct str3_typ{
UINT val4;
struct str1_typ s1;
struct str2_typ s2;
}str3_typ;

_GLOBAL str3_typ test;

All available PV Names are:
test.val4
test.s1.val1
test.s1.val2
test.s2.val3;

Top PV Name (pvNameRoot):
test

During iteration, followin values will appear for 'structItemName':
s1
s2
val4

During iteration, following values will appear for 'structItemPVNameNoRoot':
val4
s1.val1
s1.val2
s2.val3

*/
	int ii = 0;
	// TODO: checking for max size of the strings that are copied to these arrays
	char structName[256];
	char structItemName[32];
	char structItemPVNameNoRoot[256];
	UINT status;
	UDINT data_typ;
	UDINT data_len;
	UDINT adr;

	for(ii=0; ii < dimension; ii++){
		// NOTE: verify why PV_item destroys concent of the buffer supplied as 1st param
		if( !pvName){
			brsstrcpy((UDINT)structName, (UDINT)pvNameRoot);
		}else{
			brsstrcpy((UDINT)structName, (UDINT)pvNameRoot);
			brsstrcat((UDINT)structName, (UDINT)".");
			brsstrcat((UDINT)structName, (UDINT)pvName);
		}

		//DBG("1)bgPVSubStr.. ii=%d str=%s item=%s", ii, structName, structItemName);
		status = PV_item(structName, ii, structItemName);
		//DBG("2)bgPVSubStr.. ii=%d str=%s item=%s", ii, structName, structItemName);

		if(status && (status != 14713)){
			// TODO: error handling
			//DBG("bgPVSubStr.. ii=%d str=%s item=%s err=%d", ii, structName, structItemName, status);
			p->errorCode = status;
			return;
		}

		//DBG("item=%d, name=%s", ii, structItemName);
		// TODO: check for max length of the PV name
		if(!pvName){
			brsstrcpy((UDINT)structItemPVNameNoRoot, (UDINT)structItemName);
		}else{
			if(status == 14713){//14713 is to handle enum type??? find out if there is a better solutiuon
				//following code is to handle an enum type that is reported as a structure (type 0). However, there are no structure elements and is not clear how to access values???
				char pvTextValue[64];

				status = PV_ninfo(structName, &data_typ, &data_len, &dimension);
				status = PV_xgetadr(structName, &adr, &data_len);
				//based on the reported lenght, try to guess the type of the enum
				if(data_len == 1){
					data_typ = PB_DT_BYTE;
				}else
					if(data_len == 2){
					data_typ = PB_DT_WORD;
				}else{
					data_typ = PB_DT_LONG;
				}
				bgGetPVValueText(&pvTextValue[0], data_typ, data_len, dimension, adr);
				bgPVWriteOutStream(p, pvName, pvTextValue);
				return;
			}

			brsstrcpy((UDINT)structItemPVNameNoRoot, (UDINT)pvName);
			brsstrcat((UDINT)structItemPVNameNoRoot, (UDINT)".");
			brsstrcat((UDINT)structItemPVNameNoRoot, (UDINT)structItemName);
		}

		bgPVSerialize(p, pvNameRoot, structItemPVNameNoRoot);

		if(p->errorCode)
			return;
	}
}

DINT bgPVRootArraySerialize(char* pvNameRoot, char* toOutStream, UDINT lengthOutStream, UDINT begIndex, UDINT endIndex)
{
	UINT status;
	UDINT data_typ;
	UDINT data_len;
	UINT dimension;
	UDINT adr;

	bgPVSerialize_typ pvSerObj;

	if(!pvNameRoot || !toOutStream){
		return PV_SERIALIZE_ERR_ZEROPTR;
	}

	if(toOutStream){
		brsstrcpy((UDINT)toOutStream, (UDINT)"");
	}
	pvSerObj.toOutStream = toOutStream;
	pvSerObj.lengthOutStream = lengthOutStream;
	pvSerObj.outputCharCount = 0;
	pvSerObj.errorCode = 0;
	pvSerObj.arrayIndexFrom = begIndex;
	pvSerObj.arrayIndexTo = endIndex;
	pvSerObj.pItemDelim =  PV_SERIALIZE_ITEM_DELIM_COMMA;
	pvSerObj.pStrMarkup =  PV_SERIALIZE_STR_MARKUP;

	status = PV_ninfo(pvNameRoot, &data_typ, &data_len, &dimension);
	if( status ){
		return PV_SERIALIZE_ERR_PVNOTFOUND;
	}

	status = PV_xgetadr(pvNameRoot, &adr, &data_len);
	if( status ){
		return PV_SERIALIZE_ERR_PVADRNOTFOUND;
	}

	if(data_typ == PB_DT_STRUCT){
		//DBG("TOPPV='%s' Typ=%s Len=%d Dim=%d" , pvNameRoot, bgGetPVTypeString(data_typ), data_len, dimension);
		bgPVSubStructSerialize(&pvSerObj, pvNameRoot, 0, dimension);
	}else
	if(data_typ == PB_DT_ARRAY){
		bgPVArraySerializeRootToFrom(&pvSerObj, pvNameRoot, dimension);
	}
	else{
		char pvTextValue[64];
		bgGetPVValueText(&pvTextValue[0], data_typ, data_len, dimension, adr);
		//DBG("TOPPV NOT A STRUCT! PV='%s' Typ=%s Len=%d Dim=%d Val=%s" , pvNameRoot, bgGetPVTypeString(data_typ), data_len, dimension, pvTextValue);
	}

	if(pvSerObj.errorCode){
		if(pvSerObj.errorCode < 0){
			return pvSerObj.errorCode;
		}
		return (pvSerObj.errorCode * (-1));
	}

	return pvSerObj.outputCharCount;
}

DINT bgPVStructSerialize(char* pvNameRoot, char* toOutStream, UDINT lengthOutStream)
{
	UINT status;
	UDINT data_typ;
	UDINT data_len;
	UINT dimension;
	UDINT adr;
	bgPVSerialize_typ pvSerObj;

	if(!pvNameRoot || !toOutStream){
		return PV_SERIALIZE_ERR_ZEROPTR;
	}

	if(toOutStream){
		brsstrcpy((UDINT)toOutStream, (UDINT)"");
	}
	pvSerObj.toOutStream = toOutStream;
	pvSerObj.lengthOutStream = lengthOutStream;
	pvSerObj.outputCharCount = 0;
	pvSerObj.errorCode = 0;
	pvSerObj.pItemDelim =  PV_SERIALIZE_ITEM_DELIM_CRLF;
	pvSerObj.pStrMarkup =  "";

	status = PV_ninfo(pvNameRoot, &data_typ, &data_len, &dimension);
	if( status ){
		return PV_SERIALIZE_ERR_PVNOTFOUND;
	}

	status = PV_xgetadr(pvNameRoot, &adr, &data_len);
	if( status ){
		return PV_SERIALIZE_ERR_PVADRNOTFOUND;
	}

	if(data_typ == PB_DT_STRUCT){
		//DBG("TOPPV='%s' Typ=%s Len=%d Dim=%d" , pvNameRoot, bgGetPVTypeString(data_typ), data_len, dimension);
		bgPVSubStructSerialize(&pvSerObj, pvNameRoot, 0, dimension);
	}else
	if(data_typ == PB_DT_ARRAY){
		pvSerObj.arrayIndexFrom = 0;
		pvSerObj.arrayIndexTo = dimension - 1;
		bgPVArraySerializeRootToFrom(&pvSerObj, pvNameRoot, dimension);
	}
	else{
		char pvTextValue[64];
		bgGetPVValueText(&pvTextValue[0], data_typ, data_len, dimension, adr);
		//DBG("TOPPV NOT A STRUCT! PV='%s' Typ=%s Len=%d Dim=%d Val=%s" , pvNameRoot, bgGetPVTypeString(data_typ), data_len, dimension, pvTextValue);
	}

	if(pvSerObj.errorCode){
		if(pvSerObj.errorCode < 0){
			return pvSerObj.errorCode;
		}
		return (pvSerObj.errorCode * (-1));
	}

	return pvSerObj.outputCharCount;
}

//Maximum number of PV-s per file that can be deserialized!!!
#define BGPV_DESER_MAXPVCOUNT 1000

DINT bgPVStructDeserialize(char* pvNameRoot, char* fromStream, UDINT lengthStream)
{
	UDINT ii;
	bgStringListEx_typ lineList1;
	bgStringListEx_typ lineSplit1;
	char* memLineList[BGPV_DESER_MAXPVCOUNT];
	char* memLineSplit[10];
	char structItemPVName[256];

	UINT status;
	UDINT data_typ;
	UDINT data_len;
	UINT dimension;
	UDINT adr;
	UDINT errorCounter = 0;

	bgStringListLinesEx(&lineList1, fromStream, (char*)memLineList, BGPV_DESER_MAXPVCOUNT*sizeof(char*));
	for(ii=0; ii<lineList1.itemCount; ii++){
		//DBG("ln%d: %s", ii, lineList1.items[ii]);
		bgStringSplitLineEx(&lineSplit1, '=',  (char*)lineList1.items[ii], (char*)memLineSplit, (int)10*sizeof(char*));
		//DBG("ln%d: key=%s val=%s", ii, lineSplit1.items[0], lineSplit1.items[1]);

		brsstrcpy((UDINT)structItemPVName, (UDINT)pvNameRoot);
		brsstrcat((UDINT)structItemPVName, (UDINT)".");
		brsstrcat((UDINT)structItemPVName, (UDINT)lineSplit1.items[0]);

		//DBG("PV=%s Val=%s", structItemPVName, lineSplit1.items[1]);
		status = PV_ninfo(structItemPVName, &data_typ, &data_len, &dimension);

		if( status ){
			// TODO: error handling
			//DBG("bgPVStructDes. PV='%s'; Error#=%d", structItemPVName, status);
			errorCounter++;
			continue;
		}

		status = PV_xgetadr(structItemPVName, &adr, &data_len);

		if( status ){
			// TODO: error handling
			//DBG("bgPVStructDes. Address for PV='%s'; Error=%d", structItemPVName, status);
			errorCounter++;
			continue;
		}

		bgSetPVValueText((char*)lineSplit1.items[1], data_typ, data_len, dimension, adr);
	}

	// TODO: return value in case of errors; detected version changes, etc.

	return errorCounter;

}

/**
###############################################################################
###############################################################################
bgPVCompare routines
- these routines are derived/based upon the bgPVSeriliaze routines and are
used to compare two instances of the same PV type for differences
- such routine could be used, for example, when detecting a change
within a machine configuration structure or recipe
###############################################################################
###############################################################################
*/
static void bgPVArrayCompare(bgPVSerialize_typ* p, char* pvNameRoot, char* pvName, int dimension, char* pvNameRoot2)
{
	int ii = 0;
	// TODO: checking for max size of the strings that are copied to these arrays
	char structName[256];
	char structItemName[32];
	char structName2[256];
	char structItemName2[32];

	for(ii=0; ii < dimension; ii++){
		// NOTE: verify why PV_item destroys content of the buffer supplied as 1st param
		if( !pvName){
			brsstrcpy((UDINT)structName, (UDINT)pvNameRoot);
			brsstrcpy((UDINT)structName2, (UDINT)pvNameRoot2);
		}else{
			brsstrcpy((UDINT)structName, (UDINT)pvNameRoot);
			brsstrcpy((UDINT)structName2, (UDINT)pvNameRoot2);
			//strcat(structName, ".");
			//strcat(structName, pvName);
		}

		{
			char arrayIndexTxt[10];
			brsstrcpy((UDINT)structItemName, (UDINT)pvName);
			brsstrcat((UDINT)structItemName, (UDINT)"[");
			brsitoa(ii, (UDINT)arrayIndexTxt);
			brsstrcat((UDINT)structItemName, (UDINT)arrayIndexTxt);
			brsstrcat((UDINT)structItemName, (UDINT)"]");

			brsstrcpy((UDINT)structItemName2, (UDINT)pvName);
			brsstrcat((UDINT)structItemName2, (UDINT)"[");
			brsitoa(ii, (UDINT)arrayIndexTxt);
			brsstrcat((UDINT)structItemName2, (UDINT)arrayIndexTxt);
			brsstrcat((UDINT)structItemName2, (UDINT)"]");

		}

		bgPVCompare(p, structName, structItemName, structName2);

		if(p->errorCode)
			return;

	}
}

static void bgPVArrayCompareRootToFrom(bgPVSerialize_typ* p, char* pvNameRoot, int dimension, char* pvNameRoot2)
{
	int ii = 0;
	// TODO: checking for max size of the strings that are copied to these arrays
	char structItemName[32];

	char structItemName2[32];

	for(ii = p->arrayIndexFrom; (ii < dimension) && (ii <= p->arrayIndexTo); ii++){
		// NOTE: verify why PV_item destroys content of the buffer supplied as 1st param
		{
			char arrayIndexTxt[10];
			brsstrcpy((UDINT)structItemName, (UDINT)pvNameRoot);
			brsstrcat((UDINT)structItemName, (UDINT)"[");
			brsitoa(ii, (UDINT)arrayIndexTxt);
			brsstrcat((UDINT)structItemName, (UDINT)arrayIndexTxt);
			brsstrcat((UDINT)structItemName, (UDINT)"]");

			brsstrcpy((UDINT)structItemName2, (UDINT)pvNameRoot2);
			brsstrcat((UDINT)structItemName2, (UDINT)"[");
			brsitoa(ii, (UDINT)arrayIndexTxt);
			brsstrcat((UDINT)structItemName2, (UDINT)arrayIndexTxt);
			brsstrcat((UDINT)structItemName2, (UDINT)"]");

		}
		//bgTxtWriteOutStream(p, structItemName);
		//bgTxtWriteOutStream(p, "=[");
		bgPVCompare(p, structItemName, 0, structItemName2);
		//bgTxtWriteOutStream(p, "]\r\n");
		//bgTxtWriteOutStream(p, "],");

		if(p->errorCode)
			return;
	}
}

static void bgPVCompare(bgPVSerialize_typ* p, char* pvNameRoot, char* pvName, char* pvNameRoot2)
{
	UINT status;
	UDINT data_typ;
	UDINT data_len;
	UINT dimension;
	UDINT adr;
	UINT status2;
	UDINT data_typ2;
	UDINT data_len2;
	UINT dimension2;
	UDINT adr2;
	char structItemPVName[256];
	char structItemPVName2[256];

	if( !pvName){
		brsstrcpy((UDINT)structItemPVName, (UDINT)pvNameRoot);
		brsstrcpy((UDINT)structItemPVName2, (UDINT)pvNameRoot2);

	}else{
		brsstrcpy((UDINT)structItemPVName, (UDINT)pvNameRoot);
		brsstrcat((UDINT)structItemPVName, (UDINT)".");
		brsstrcat((UDINT)structItemPVName, (UDINT)pvName);

		brsstrcpy((UDINT)structItemPVName2, (UDINT)pvNameRoot2);
		brsstrcat((UDINT)structItemPVName2, (UDINT)".");
		brsstrcat((UDINT)structItemPVName2, (UDINT)pvName);
	}

	status = PV_ninfo(structItemPVName, &data_typ, &data_len, &dimension);
	status2 = PV_ninfo(structItemPVName2, &data_typ2, &data_len2, &dimension2);

	if( status ){
		p->errorCode = status;
		return;
	}
	if( status2 ){
		p->errorCode = status2;
		return;
	}

	if( bgPVSerializeIsArray(data_typ, data_len, dimension) ){
		bgPVArrayCompare(p, pvNameRoot, pvName, dimension, pvNameRoot2);
		return;
	}

	status = PV_xgetadr(structItemPVName, &adr, &data_len);
	status2 = PV_xgetadr(structItemPVName2, &adr2, &data_len2);

	if( status ){
		p->errorCode = status;
		return;
	}
	if( status2 ){
		p->errorCode = status2;
		return;
	}

	if(data_typ == PB_DT_STRUCT){
		//DBG("PV='%s' Typ=%s Len=%d Dim=%d" , pvnamecomplete, bgGetPVTypeString(data_typ), data_len, dimension);
		bgPVSubStructCompare(p, pvNameRoot, pvName, dimension, pvNameRoot2);
	}else{
		char pvTextValue[256];
		char pvTextValue2[256];
		int len = 0;

		if(data_typ == PB_DT_VIS){//STRING VALUES ONLY > marked with a special markup at the begining and end
			brsstrcpy((UDINT)pvTextValue, (UDINT)p->pStrMarkup);//set string begining markup (i.e. "\"")
			brsstrcpy((UDINT)pvTextValue2, (UDINT)p->pStrMarkup);//set string begining markup (i.e. "\"")
			len = brsstrlen((UDINT)pvTextValue);
		}

		bgGetPVValueText(&pvTextValue[len], data_typ, data_len, dimension, adr);
		bgGetPVValueText(&pvTextValue2[len], data_typ2, data_len2, dimension2, adr2);

		if(data_typ == PB_DT_VIS){//STRING VALUES ONLY > marked with a special markup at the begining and end
			brsstrcat((UDINT)pvTextValue, (UDINT)p->pStrMarkup);//set string ending markup (i.e. "\"")
			brsstrcat((UDINT)pvTextValue2, (UDINT)p->pStrMarkup);//set string ending markup (i.e. "\"")
		}

		if(brsstrcmp((UDINT)pvTextValue, (UDINT)pvTextValue2) != 0){
			char buf[255];
			sprintf2(buf, "%s changed; Old=%s, New=%s\n", structItemPVName, pvTextValue2, pvTextValue);
			bgTxtWriteOutStream(p, buf);
		}

		//DBG("stritemPV='%s' Typ=%s Len=%d Dim=%d Val=%s" , pvName, bgGetPVTypeString(data_typ), data_len, dimension, pvTextValue);
		//bgPVWriteOutStream(p, pvName, pvTextValue);
	}

}

static void bgPVSubStructCompare(bgPVSerialize_typ* p, char* pvNameRoot, char* pvName, UINT dimension, char* pvNameRoot2)
{

	int ii = 0;
	// TODO: checking for max size of the strings that are copied to these arrays
	char structName[256];
	char structName2[256];
	char structItemName[32];
	char structItemName2[32];
	char structItemPVNameNoRoot[256];
	char structItemPVNameNoRoot2[256];
	UINT status;
	UINT status2;
	UDINT data_typ;
	UDINT data_typ2;
	UDINT data_len;
	UDINT data_len2;
	UDINT adr;
	UDINT adr2;
	UINT dimension2;

	for(ii=0; ii < dimension; ii++){
		// NOTE: verify why PV_item destroys concent of the buffer supplied as 1st param
		if( !pvName){
			brsstrcpy((UDINT)structName, (UDINT)pvNameRoot);
			brsstrcpy((UDINT)structName2, (UDINT)pvNameRoot2);
		}else{
			brsstrcpy((UDINT)structName, (UDINT)pvNameRoot);
			brsstrcat((UDINT)structName, (UDINT)".");
			brsstrcat((UDINT)structName, (UDINT)pvName);

			brsstrcpy((UDINT)structName2, (UDINT)pvNameRoot2);
			brsstrcat((UDINT)structName2, (UDINT)".");
			brsstrcat((UDINT)structName2, (UDINT)pvName);
		}

		status = PV_item(structName, ii, structItemName);
		status2 = PV_item(structName2, ii, structItemName2);

		if(status && (status != 14713)){
			// TODO: error handling
			//DBG("bgPVSubStr.. ii=%d str=%s item=%s err=%d", ii, structName, structItemName, status);
			p->errorCode = status;
			return;
		}
		if(status2 && (status2 != 14713)){
			// TODO: error handling
			//DBG("bgPVSubStr.. ii=%d str=%s item=%s err=%d", ii, structName, structItemName, status);
			p->errorCode = status2;
			return;
		}

		//DBG("item=%d, name=%s", ii, structItemName);
		// TODO: check for max length of the PV name
		if(!pvName){
			brsstrcpy((UDINT)structItemPVNameNoRoot, (UDINT)structItemName);
			brsstrcpy((UDINT)structItemPVNameNoRoot2, (UDINT)structItemName2);
		}else{
			if(status == 14713){//14713 is to handle enum type??? find out if there is a better solutiuon
				//following code is to handle an enum type that is reported as a structure (type 0). However, there are no structure elements and is not clear how to access values???
				char pvTextValue[64];
				char pvTextValue2[64];

				status = PV_ninfo(structName, &data_typ, &data_len, &dimension);
				status = PV_xgetadr(structName, &adr, &data_len);

				status2 = PV_ninfo(structName2, &data_typ2, &data_len2, &dimension2);
				status2 = PV_xgetadr(structName2, &adr2, &data_len2);

				//based on the reported lenght, try to guess the type of the enum
				if(data_len == 1){
					data_typ = PB_DT_BYTE;
				}else
					if(data_len == 2){
					data_typ = PB_DT_WORD;
				}else{
					data_typ = PB_DT_LONG;
				}
				bgGetPVValueText(&pvTextValue[0], data_typ, data_len, dimension, adr);
				bgGetPVValueText(&pvTextValue2[0], data_typ2, data_len2, dimension2, adr2);
				if(brsstrcmp((UDINT)&pvTextValue[0], (UDINT)&pvTextValue2[0]) != 0){
					char buf[255];
					sprintf2(buf, "%s changed; Old=%s, New=%s\n", structName, &pvTextValue2[0], &pvTextValue[0]);
					bgTxtWriteOutStream(p, buf);
				}
				return;
			}

			brsstrcpy((UDINT)structItemPVNameNoRoot, (UDINT)pvName);
			brsstrcat((UDINT)(UDINT)structItemPVNameNoRoot, (UDINT)".");
			brsstrcat((UDINT)(UDINT)structItemPVNameNoRoot, (UDINT)structItemName);

			brsstrcpy((UDINT)structItemPVNameNoRoot2, (UDINT)pvName);
			brsstrcat((UDINT)structItemPVNameNoRoot2, (UDINT)".");
			brsstrcat((UDINT)structItemPVNameNoRoot2, (UDINT)structItemName2);

		}

		bgPVCompare(p, pvNameRoot, structItemPVNameNoRoot, pvNameRoot2);

		if(p->errorCode)
			return;
	}
}

DINT bgPVRootArrayCompare(char* pvNameRoot, char* toOutStream, UDINT lengthOutStream, UDINT begIndex, UDINT endIndex, char* pvNameRoot2)
{
	UINT status;
	UDINT data_typ;
	UDINT data_len;
	UINT dimension;
	UDINT adr;

	bgPVSerialize_typ pvSerObj;

	if(!pvNameRoot || !toOutStream){
		return PV_SERIALIZE_ERR_ZEROPTR;
	}

	if(toOutStream){
		brsstrcpy((UDINT)toOutStream, (UDINT)"");
	}
	pvSerObj.toOutStream = toOutStream;
	pvSerObj.lengthOutStream = lengthOutStream;
	pvSerObj.outputCharCount = 0;
	pvSerObj.errorCode = 0;
	pvSerObj.arrayIndexFrom = begIndex;
	pvSerObj.arrayIndexTo = endIndex;
	pvSerObj.pItemDelim =  PV_SERIALIZE_ITEM_DELIM_COMMA;
	pvSerObj.pStrMarkup =  PV_SERIALIZE_STR_MARKUP;

	status = PV_ninfo(pvNameRoot, &data_typ, &data_len, &dimension);
	if( status ){
		return PV_SERIALIZE_ERR_PVNOTFOUND;
	}

	status = PV_xgetadr(pvNameRoot, &adr, &data_len);
	if( status ){
		return PV_SERIALIZE_ERR_PVADRNOTFOUND;
	}

	if(data_typ == PB_DT_STRUCT){
		//DBG("TOPPV='%s' Typ=%s Len=%d Dim=%d" , pvNameRoot, bgGetPVTypeString(data_typ), data_len, dimension);
		bgPVSubStructCompare(&pvSerObj, pvNameRoot, 0, dimension, pvNameRoot2);
	}else
	if(data_typ == PB_DT_ARRAY){
		bgPVArrayCompareRootToFrom(&pvSerObj, pvNameRoot, dimension, pvNameRoot2);
	}
	else{
		char pvTextValue[64];
		bgGetPVValueText(&pvTextValue[0], data_typ, data_len, dimension, adr);
		//DBG("TOPPV NOT A STRUCT! PV='%s' Typ=%s Len=%d Dim=%d Val=%s" , pvNameRoot, bgGetPVTypeString(data_typ), data_len, dimension, pvTextValue);
	}

	if(pvSerObj.errorCode){
		if(pvSerObj.errorCode < 0){
			return pvSerObj.errorCode;
		}
		return (pvSerObj.errorCode * (-1));
	}

	return pvSerObj.outputCharCount;
}

DINT bgPVStructCompare(char* pvNameRoot, char* pvNameRoot2, char* toOutStream, UDINT lengthOutStream)
{
	UINT status;
	UDINT data_typ, data_typ2;
	UDINT data_len, data_len2;
	UINT dimension, dimension2;
	UDINT adr, adr2;
	bgPVSerialize_typ pvSerObj;

	if(!pvNameRoot || !pvNameRoot2 || !toOutStream){
		return PV_SERIALIZE_ERR_ZEROPTR;
	}

	if(toOutStream){
		brsstrcpy((UDINT)toOutStream, (UDINT)"");
	}
	pvSerObj.toOutStream = toOutStream;
	pvSerObj.lengthOutStream = lengthOutStream;
	pvSerObj.outputCharCount = 0;
	pvSerObj.errorCode = 0;
	pvSerObj.pItemDelim =  PV_SERIALIZE_ITEM_DELIM_CRLF;
	pvSerObj.pStrMarkup =  "";

	status = PV_ninfo(pvNameRoot, &data_typ, &data_len, &dimension);
	if( status ){
		return PV_SERIALIZE_ERR_PVNOTFOUND;
	}
	status = PV_xgetadr(pvNameRoot, &adr, &data_len);
	if( status ){
		return PV_SERIALIZE_ERR_PVADRNOTFOUND;
	}

	status = PV_ninfo(pvNameRoot2, &data_typ2, &data_len2, &dimension2);
	if( status ){
		return PV_SERIALIZE_ERR_PVNOTFOUND;
	}
	status = PV_xgetadr(pvNameRoot2, &adr2, &data_len2);
	if( status ){
		return PV_SERIALIZE_ERR_PVADRNOTFOUND;
	}

	//struct must be equvalenet to compare them
	if((data_typ != data_typ2) || (dimension != dimension2) || (data_len != data_len2)){
		return PV_SERIALIZE_ERR_NOCOMPARE;
	}

	if(data_typ == PB_DT_STRUCT){
		//DBG("TOPPV='%s' Typ=%s Len=%d Dim=%d" , pvNameRoot, bgGetPVTypeString(data_typ), data_len, dimension);
		bgPVSubStructCompare(&pvSerObj, pvNameRoot, 0, dimension, pvNameRoot2);
	}else
	if(data_typ == PB_DT_ARRAY){
		pvSerObj.arrayIndexFrom = 0;
		pvSerObj.arrayIndexTo = dimension - 1;
		bgPVArrayCompareRootToFrom(&pvSerObj, pvNameRoot, dimension, pvNameRoot2);
	}
	else{
		char pvTextValue[64];
		bgGetPVValueText(&pvTextValue[0], data_typ, data_len, dimension, adr);
		//DBG("TOPPV NOT A STRUCT! PV='%s' Typ=%s Len=%d Dim=%d Val=%s" , pvNameRoot, bgGetPVTypeString(data_typ), data_len, dimension, pvTextValue);
	}

	if(pvSerObj.errorCode){
		if(pvSerObj.errorCode < 0){
			return pvSerObj.errorCode;
		}
		return (pvSerObj.errorCode * (-1));
	}

	return pvSerObj.outputCharCount;
}

#endif //_BG_SERIALIZE_C
/*EOF*/
```

### bgTelnetSrvr-astcpV2.h
```c
#include <bur/plctypes.h>
#ifndef _BG_TELNETSERVER_V2_H
#define _BG_TELNETSERVER_V2_H

#ifdef _DEFAULT_INCLUDES
	#include <AsDefault.h>
#endif

#include "bgringbuffer.h"

void bgTelnetSrvrInit(bgSocketServer_typ* pTerm, bgRingBuffer_typ* pRB);

void bgTelnetSrvrCyclic(bgSocketServer_typ* pTerm);

#endif
```

### Program Logical/paiComponents/LibAsUSB1_ST/read_data

#### read_data.var
```iecst
(********************************************************************
 * COPYRIGHT -- Bernecker + Rainer
 ********************************************************************
 * Program: read_data
 * File: read_data.var
 * Author: Bernecker & Rainer
 * Created: April 20, 2009
 ********************************************************************
 * Local variables of program read_data
 ********************************************************************)
VAR CONSTANT
	CREATE_NODE_ID_LIST : USINT := 2; (*Function step: Create a list of Node-IDs from all active USB devices*)
	READ_DEVICE_DATA : USINT := 3; (*Function step: Read out the specific data from the Node-IDs*)
	GET_DESCRIPTOR : USINT := 4; (*Function step: Read out the descriptor data from the Node-IDs*)
	CREATE_FILE_DEVICE : USINT := 5; (*Function step: Create file out of data from USB device*)
	DIRECTORY_READ : USINT := 7; (*Function step: Read out to data from linked File Device*)
	UNLINK_DEVICE : USINT := 9; (*Function step: Unlink the File Device from specific path*)
	FINISH : USINT := 8; (*Function step: Function chain is finished - back to WAIT*)
	WAIT : USINT := 0; (*Function step: Wait for starting the Function chain*)
	DIRECTORY_INFO : USINT := 6; (*Function step: Read out the Info about the connected File Device*)
	ERROR_CASE : USINT := 1; (*Function step: Jump to this step in every case of Error occuring in the Function chain*)
END_VAR
VAR
	device_data : fiDIR_READ_DATA := (0); (*Buffer to store device data*)
	device_descriptor : ARRAY[0..4] OF usbDeviceDescr_typ; (*Buffer to store descriptor data of device*)
	usb_data_buffer : ARRAY[0..4] OF usbNode_typ; (*Defined data_typ of AsUSB - Library*)
	node_id_buffer : ARRAY[0..4] OF UDINT; (*Different nodeIDs saved in array-elements*)
	UsbNodeListGet_0 : UsbNodeListGet; (*Type of FUB UsbNodeListGet*)
	step : USINT; (*Determines the Function step*)
	UsbNodeGet_0 : UsbNodeGet; (*Type of FUB UsbNodeGet*)
	start_reading_usb_data : BOOL; (*If TRUE - Function chain gets started*)
	node : USINT; (*Node number*)
	DevLink_0 : DevLink; (*Type of FUB DevLink*)
	UsbDescriptorGet_0 : UsbDescriptorGet; (*Type of FUB UsbDescriptorGet*)
	device_name : STRING[80]; (*Name of the USB device - optional *)
	device_param : STRING[80]; (*Connection path of USB device*)
	DirInfo_0 : DirInfo; (*Type of FUB DirInfo*)
	DirRead_0 : DirRead; (*Type of FUB DirRead*)
	DevUnlink_0 : DevUnlink; (*Type of FUB DevUnlink*)
END_VAR
```

#### read_data.st
```iecst
(********************************************************************
 * COPYRIGHT -- Bernecker + Rainer
 ********************************************************************
 * Program: read_data
 * File: read_data.st
 * Author: Bernecker & Rainer
 * Created: April 20, 2009
 ********************************************************************
 * Implementation of program read_data
 ********************************************************************)

PROGRAM _INIT

	step := WAIT;

END_PROGRAM

PROGRAM _CYCLIC

CASE step OF

	WAIT:

		IF start_reading_usb_data = TRUE THEN
			step := CREATE_NODE_ID_LIST;  (*start FUBs below*)
		ELSE
			step := WAIT;
		END_IF;

	CREATE_NODE_ID_LIST:  (*Library AsUSB - Functionblock USBNodeListGet()*)

		UsbNodeListGet_0.enable := 1;
		UsbNodeListGet_0.pBuffer := ADR(node_id_buffer);  (*pointer to buffer - UDINT array is assigned*)
		UsbNodeListGet_0.bufferSize := SIZEOF(node_id_buffer);  (*size of node-id-buffer-array*)
		UsbNodeListGet_0.filterInterfaceClass := 0;//asusb_CLASS_MASS_STORAGE;  (*filter on mass storage devices is set*)
		UsbNodeListGet_0.filterInterfaceSubClass := 0;  (*no filer is set*)
		UsbNodeListGet_0;

		IF UsbNodeListGet_0.status = 0 THEN
        	step := READ_DEVICE_DATA;  (*FUB worked correctly => next step*)
		ELSIF UsbNodeListGet_0.status = ERR_FUB_BUSY THEN
			step := CREATE_NODE_ID_LIST;  (*FUB work asynchron => called until status isn't BUSY*)
		ELSE
			step := ERROR_CASE;  (*error occured*)
		END_IF;

	READ_DEVICE_DATA:  (*Library AsUSB - Functionblock USBNodeGet()*)

		UsbNodeGet_0.enable := 1;
		UsbNodeGet_0.nodeId := node_id_buffer[node];  (*specific node is read out of node_id_buffer*)
		UsbNodeGet_0.pBuffer := ADR(usb_data_buffer[node]);  (*data of specific node get stored in usb_data_buffer*)
		UsbNodeGet_0.bufferSize := SIZEOF (usb_data_buffer[node]);  (*size of specific node is read out usb_data_buffer*)
		UsbNodeGet_0;

		IF UsbNodeGet_0.status = 0 THEN  (*FUB worked correctly*)
			node := node + 1;  (*next node to be read out of buffer*)
			IF node = UsbNodeListGet_0.listNodes THEN  (*last existing node is reached*)
				node := 0;
				step := GET_DESCRIPTOR;  (*all nodes are read out of buffer*)
			END_IF;

		ELSIF UsbNodeGet_0.status = ERR_FUB_BUSY THEN
			step := READ_DEVICE_DATA;  (*FUB work asynchron => called until status isn't BUSY*)
		ELSE
			step := ERROR_CASE;  (*error occured*)
		END_IF;

	GET_DESCRIPTOR:  (*Library AsUSB - Functionblock USBDescriptorGet()*)

		UsbDescriptorGet_0.enable := 1;
		UsbDescriptorGet_0.nodeId := node_id_buffer[node];  (*specific node is read out of node_id_buffer*)
		UsbDescriptorGet_0.requestType := 0;  (*Request for device*)
        UsbDescriptorGet_0.descriptorType := 1;  (*Determines the device descriptor*)
		UsbDescriptorGet_0.languageId := 0;  (*for device and configuration descriptors*)
		UsbDescriptorGet_0.pBuffer := ADR(device_descriptor[node]);  (*descriptor-data of specific node get stored in device_descriptor-buffer*)
		UsbDescriptorGet_0.bufferSize := SIZEOF(device_descriptor[node]);  (*size of specific node is read out device_descriptor-buffer*)
		UsbDescriptorGet_0;

		IF UsbDescriptorGet_0.status = 0 THEN  (*FUB worked correctly*)
			node := node + 1;  (*next node to be read out of buffer*)
			IF node = UsbNodeListGet_0.listNodes THEN  (*last existing node is reached*)
				node := 0;
				step := CREATE_FILE_DEVICE;  (*all nodes are read out of buffer*)
			END_IF;

		ELSIF UsbDescriptorGet_0.status = ERR_FUB_BUSY THEN
			step := GET_DESCRIPTOR;  (*FUB work asynchron => called until status isn't BUSY*)
		ELSE
			step := ERROR_CASE;  (*error occured*)
		END_IF;

	CREATE_FILE_DEVICE:  (*Library FileIO - Functionblock DevLink() - create file out of data just from 1. USB*)

		strcpy(ADR(device_name), ADR('DEVICE1'));  (*fixed Device-Name get copied to device_name-Variable*)
		strcpy(ADR(device_param), ADR('/DEVICE='));  (*first part of parameter get copied to device_param-Variable*)
		strcat(ADR(device_param), ADR(usb_data_buffer[0].ifName));  (*second part get added to device_param-Variable*)

		DevLink_0.enable := 1;
		DevLink_0.pDevice := ADR(device_name);  (*Devicename is assigned*)
		DevLink_0.pParam := ADR(device_param);  (*the path of the Device is assigned*)
		DevLink_0;

		IF DevLink_0.status = 0 THEN
			step := DIRECTORY_INFO;  (*FUB worked correctly => next step*)
		ELSIF DevLink_0.status = ERR_FUB_BUSY THEN
			step := CREATE_FILE_DEVICE;  (*FUB work asynchron => called until status isn't BUSY*)
		ELSE
			step := ERROR_CASE;  (*error occured*)
		END_IF;

	DIRECTORY_INFO:  (*Library FileIO - Functionblock DirInfo()*)

		DirInfo_0.enable := 1;
		DirInfo_0.pDevice := ADR(device_name);  (*Devicename is assigned*)
		DirInfo_0.pPath := 0;  (*no path is needed => value = 0*)
		DirInfo_0;

		IF DirInfo_0.status = 0 THEN
			step := DIRECTORY_READ;  (*FUB worked correctly => next step*)
		ELSIF DirInfo_0.status = ERR_FUB_BUSY THEN
			step := DIRECTORY_INFO;  (*FUB work asynchron => called until status isn't BUSY*)
		ELSE
			step := ERROR_CASE;  (*error occured*)
		END_IF;

	DIRECTORY_READ:  (*Library FileIO - Functionblock DirRead()*)

		DirRead_0.enable := 1;
		DirRead_0.pDevice := ADR(device_name);  (*Devicename is assigned*)
		DirRead_0.pPath := 0;  (*no path is needed => value = 0*)
		DirRead_0.entry := 1;  (*only the first entry is read out*)
		DirRead_0.option := fiBOTH;  (*Collect information from files and directories*)
		DirRead_0.pData := ADR(device_data);  (*device_data-variable with fiDIR_READ_DATA type is assigned to data-buffer*)
		DirRead_0.data_len := SIZEOF(device_data); (*size of device_data-variable is read out*)
		DirRead_0;

		IF DirRead_0.status = 0 THEN
			step := UNLINK_DEVICE;  (*FUB worked correctly => next step*)
		ELSIF DirRead_0.status = ERR_FUB_BUSY THEN
			step := DIRECTORY_READ;  (*FUB work asynchron => called until status isn't BUSY*)
		ELSE
			step := ERROR_CASE;  (*error occured*)
		END_IF;

	UNLINK_DEVICE:  (*Library FileIO - Functionblock DevUnlink()*)

		DevUnlink_0.enable := 1;
		DevUnlink_0.handle := DevLink_0.handle;  (*handle from DevLink is assigned to cut the connection to specific file-device*)
		DevUnlink_0;

		IF DevUnlink_0.status = 0 THEN
			step := FINISH;  (*FUB worked correctly => next step*)
		ELSIF DevUnlink_0.status = ERR_FUB_BUSY THEN
			step := UNLINK_DEVICE;  (*FUB work asynchron => called until status isn't BUSY*)
		ELSE
			step := ERROR_CASE;  (*error occured*)
		END_IF;

	FINISH:  (*successfully finished*)

		start_reading_usb_data := FALSE;
		step := WAIT;  (*back to beginning - wait for start_reading_usb_data to be set*)

	ERROR_CASE:	(*error-handling*)

END_CASE;

END_PROGRAM
```

### Library Logical/paiComponents/Libraries/bglibas (ANSIC) - Simple state machine support
Depends on: standard

#### bglibas.fun
```iecst
(********************************************************************
 * COPYRIGHT -- pai
 ********************************************************************
 * Library: bglibas
 * File: bglibas.fun
 * Author: admin
 * Created: March 07, 2012
 ********************************************************************
 * Functions and function blocks of library bglibas
 ********************************************************************)
(*=========================================================================*)
(*SUPPORT FOR SIMPLE STATE MACHINE (SSM)*)
(*=========================================================================*)

FUNCTION bgSSMInit : UDINT (*Init state machine. MUST be called once, before any other bgSSM function call.*)
	VAR_INPUT
		p : bgSSM_typ;
		pfunGetStateName : UDINT;
		pfunCyclicCallback : UDINT;
	END_VAR
END_FUNCTION

FUNCTION bgSSMCyclic : UDINT (*State machine cyclic operation.*)
	VAR_INPUT
		p : bgSSM_typ;
	END_VAR
END_FUNCTION

FUNCTION bgSSMStateNextTimeDelay : UDINT (*Set SM next state w. timer delay*)
	VAR_INPUT
		p : bgSSM_typ;
		stateNext : UDINT;
		timeDelayX1ms : UDINT;
	END_VAR
END_FUNCTION

FUNCTION bgSSMStateNextCycleDelay : UDINT (*Set SM next state w. cycles delay*)
	VAR_INPUT
		p : bgSSM_typ;
		stateNext : UDINT;
		delayCycles : UDINT;
	END_VAR
END_FUNCTION

FUNCTION bgSSMStateNext : UDINT (*Set SM next state.*)
	VAR_INPUT
		p : bgSSM_typ;
		stateNext : UDINT;
	END_VAR
END_FUNCTION

FUNCTION bgSSMIsStateInit : BOOL (*Check if first scan within the current state.*)
	VAR_INPUT
		p : bgSSM_typ;
	END_VAR
END_FUNCTION

FUNCTION bgSSMGetState : UDINT (*Get current SM state*)
	VAR_INPUT
		p : bgSSM_typ;
	END_VAR
END_FUNCTION

FUNCTION bgSSMGetStateText : STRING[32] (*Get current SM state name*)
	VAR_INPUT
		p : bgSSM_typ;
	END_VAR
END_FUNCTION
(*=========================================================================*)
(*SUPPORT FOR FIFOs*)
(*=========================================================================*)

FUNCTION bgFIFOInit : UDINT (*Init simple FIFO. Stores upto (entryTotalCount) number of elements. Elements MUST be of the same size.*)
	VAR_INPUT
		p : bgFIFO_typ;
		entrySize : UDINT;
		entryTotalCount : UDINT;
		pFIFOmem : UDINT;
	END_VAR
END_FUNCTION

FUNCTION bgFIFOPush : UDINT (*Push data to FIFO. Content from pSrc is copied into the available FIFO memory. In case of error return value is != 0*)
	VAR_INPUT
		p : bgFIFO_typ;
		pSrc : UDINT;
		srcSize : UDINT;
	END_VAR
END_FUNCTION

FUNCTION bgFIFOPull : UDINT (*Pull (retrive) data from FIFO. Oldest entry from FIFO memory is copied into the provided pDst space. In case of error return value is != 0*)
	VAR_INPUT
		p : bgFIFO_typ;
		pDst : UDINT;
		dstSize : UDINT;
	END_VAR
END_FUNCTION

FUNCTION bgFIFOGetCount : UDINT (*Get number of entries stored in the FIFO*)
	VAR_INPUT
		p : bgFIFO_typ;
	END_VAR
END_FUNCTION

FUNCTION bgFIFOIsFull : UDINT (*Check if FIFO is full*)
	VAR_INPUT
		p : bgFIFO_typ;
	END_VAR
END_FUNCTION
(*=========================================================================*)
(*Support for TIMERs*)
(*=========================================================================*)

FUNCTION bgTimerCyclic : UDINT (*Timer cyclic function. Must be called cyclicly for corret timer operation.*)
	VAR_INPUT
		pTON : TON;
	END_VAR
END_FUNCTION

FUNCTION bgTimerStart : UDINT (*Start timer for a defined amount of time [ms]. IMPORTANT: function uses TON library call. Same restrictions apply!*)
	VAR_INPUT
		pTON : TON;
		timeoutTimeX1ms : UDINT;
	END_VAR
END_FUNCTION

FUNCTION bgTimerStop : UDINT (*Stop the timer.*)
	VAR_INPUT
		pTON : TON;
	END_VAR
END_FUNCTION

FUNCTION bgTimerIsEnabled : BOOL (*Check if timer is enabled.*)
	VAR_INPUT
		pTON : TON;
	END_VAR
END_FUNCTION

FUNCTION bgTimerIsTimeOut : BOOL (*Check if timer has expired.*)
	VAR_INPUT
		pTON : TON;
	END_VAR
END_FUNCTION

FUNCTION bgTimerTimeElapsed : UDINT (*Retrive the elapsed timer time [ms]*)
	VAR_INPUT
		pTON : TON;
	END_VAR
END_FUNCTION

FUNCTION bgTimerTimeRemaining : UDINT (*Retrive the remainig timer time [ms]*)
	VAR_INPUT
		pTON : TON;
	END_VAR
END_FUNCTION
```

#### bgssm.c
```c
/********************************************************************
 * COPYRIGHT -- pai
 ********************************************************************
 * Library: bglibas
 * File: bglibas.c
 * Author: admin
 * Created: March 07, 2012
 ********************************************************************
 * Implementation of library bglibas
 ********************************************************************/

#include <bur/plctypes.h>
#ifdef __cplusplus
	extern "C"
	{
#endif

#include "bglibas.h"

#ifdef __cplusplus
	};
#endif

#include <AsBrStr.h>

/* Init state machine. MUST be called once, before any other bgSSM function call. */
unsigned long bgSSMInit(struct bgSSM_typ* p, unsigned long pFunGetStateName, unsigned long pFunCyclicCallback)
{
	/*TODO: Add your code here*/
	brsmemset((UDINT)p, 0, sizeof(struct bgSSM_typ));

	p->pfunGetStateName = (UDINT)pFunGetStateName;
	p->pfunCyclicCallback = (UDINT)pFunCyclicCallback;
	p->stateInit = 1;
	return(0);
}
/* State machine cyclic operation. */
unsigned long bgSSMCyclic(struct bgSSM_typ* p)
{
	/*TODO: Add your code here*/
	int ii;

	//operate all timers
	for(ii=0; ii<BGSSM_TIMER_COUNT;ii++){
		bgTimerCyclic(&p->timer_x1ms[ii]);
	}
	bgTimerCyclic(&p->dlytimer_x1ms);

	//operate dlyCycle counter
	if(p->dlyCycles){
		p->dlyCycles--;
	}

	//call cyclic callback function if defined
	if(p->pfunCyclicCallback){
		void(*callback)(bgSSM_typ*) = ( void (*) (bgSSM_typ*) ) p->pfunCyclicCallback;
		(*callback)(p);
	}

	//clear single cycle flag every scan
	p->stateInit = 0;

	//check if state change requested
	if(p->state != p->stateNext){

		//if state change w. delay > wait for delay timer to expire or dlyCycles == 0
		if(!bgTimerIsTimeOut(&p->dlytimer_x1ms) || p->dlyCycles){
			return 1;
		}

		p->state = p->stateNext;
		//generate stateInit sigle scan flag
		p->stateInit = 1;

		//define state name if exteranl function for state names is defined
		if( p->pfunGetStateName ){
			char*(*getStateName)(UDINT) = ( char* (*) (UDINT) )p->pfunGetStateName;
			brsstrcpy((UDINT)p->stateText, (UDINT)((*getStateName)(p->state)));
		}else{
			brsstrcpy((UDINT)p->stateText, (UDINT)"???");
		}
	}
	return(0);
}
/* Change to next state. */
unsigned long bgSSMStateNext(struct bgSSM_typ* p, unsigned long stateNext)
{
	/*TODO: Add your code here*/
	p->stateNext = stateNext;
	return(p->stateNext);
}

/* Change to next state w. timer delay. */
unsigned long bgSSMStateNextTimeDelay(struct bgSSM_typ* p, unsigned long stateNext, unsigned long delayTimeX1ms)
{
	/*TODO: Add your code here*/
	p->stateNext = stateNext;
	bgTimerStart(&p->dlytimer_x1ms, delayTimeX1ms);
	return(p->stateNext);
}

/* Change to next state w. cycles delay. */
unsigned long bgSSMStateNextCycleDelay(struct bgSSM_typ* p, unsigned long stateNext, unsigned long delayCycles)
{
	/*TODO: Add your code here*/
	p->stateNext = stateNext;
	p->dlyCycles = delayCycles;
	return(p->stateNext);
}
/* Check if first scan for the state. */
plcbit bgSSMIsStateInit(struct bgSSM_typ* p)
{
	/*TODO: Add your code here*/
	return(p->stateInit);
}
//EOF

/* Get current state */
unsigned long bgSSMGetState(struct bgSSM_typ* p)
{
	/*TODO: Add your code here*/
	return(p->state);
}

/* Get current state text*/
plcstring* bgSSMGetStateText(struct bgSSM_typ* p)
{
	/*TODO: Add your code here*/
	return(&p->stateText[0]);
}
```

#### bgfifo.c
```c
/********************************************************************
 * COPYRIGHT -- HP
 ********************************************************************
 * Library: bglibas
 * File: bgfifo.c
 * Author: goran
 * Created: February 01, 2013
 *******************************************************************/

#include <bur/plctypes.h>
#ifdef __cplusplus
	extern "C"
	{
#endif

#include "bglibas.h"

#ifdef __cplusplus
	};
#endif
#include <string.h>

static void bgFIFOPushEntry(bgFIFO_typ* p)
{
	char *pSrc = (char*)p->iPtrPushData;//src data
	char* pDst = (char*)((char*)p->prvFIFOMemory + (p->cfgEntrySize * p->oPushIdx));//empty FIFO location
	memcpy(pDst, pSrc, p->cfgEntrySize);

	p->oPushIdx++;//inc location index to next empty FIFO spot
	if(p->oPushIdx >= p->cfgMaxEntries){
		p->oPushIdx = 0;//handle roll over (ring buffer)
	}

	p->oFIFOCount++;//inc number of FIFO entries
	if(p->oFIFOCount >= p->cfgMaxEntries){
		p->oFIFOFull = 1;//set FIFO full indication
	}
}

static void bgFIFOPullEntry(bgFIFO_typ* p)
{
	char* pSrc = (char*)((char*)p->prvFIFOMemory + (p->cfgEntrySize * p->oPullIdx));//oldest FIFO entry
	char *pDst = (char*)p->oPtrPullData;//destination
	memcpy(pDst, pSrc, p->cfgEntrySize);

	p->oPullIdx++;//inc oldest stored FIFO entry position
	if(p->oPullIdx >= p->cfgMaxEntries){
		p->oPullIdx = 0;//handle roll over (ring buffer)
	}

	if(p->oFIFOCount)//dec number of entris in the FIFO
		p->oFIFOCount--;

	p->oFIFOFull = 0;//reset FIFO full indication
}

/**
bgFIFOInit()
-simple FIFO. Stores upto (entryTotalCount) number of elements. Elements MUST be of the same size.
-supports push/pull action
-push:
- user supplied data is copied into the available FIFO memory space, number of items in the FIFO gets incremented,
index variable that keeps track of next empty FIFO location is adjusted; if FIFO full - no action, error returned
-pull:
- oldest entry from FIFO copied to user supplied data space; number of items in the FIFO gets decremented,
index variable that keeps track of oldeset FIFO entry is adjusted; if FIFO empty - no action, error is returned
*/
unsigned long bgFIFOInit(struct bgFIFO_typ* p, unsigned long  entrySize, unsigned long  entryTotalCount, unsigned long  pFIFOMem)
{
	if(!p || !pFIFOMem || !entrySize || (entryTotalCount <=5))
		return 1;

	p->iPtrPushData = 0;
	p->oPtrPullData = 0;

	p->oFIFOCount = 0;
	p->oFIFOFull = 0;

	p->cfgEntrySize = entrySize;
	p->cfgMaxEntries = entryTotalCount;
	p->prvFIFOMemory = pFIFOMem;
	p->oPullIdx = 0;
	p->oPushIdx = 0;
	return 0;
}

/* Push data to FIFO. Content from pSrc is copied into the available FIFO memory. In case of error return value is != 0*/
unsigned long bgFIFOPush(struct bgFIFO_typ* p, unsigned long pSrc, unsigned long srcSize)
{
	if(!p)
		return 1;

	if(!p->prvFIFOMemory)
		return 2;

	if(!pSrc)
		return 3;

	if(!srcSize || (srcSize != p->cfgEntrySize) )
		return 4;

	if(p->oFIFOFull)
		return 5;

	p->iPtrPushData = pSrc;
	bgFIFOPushEntry(p);
	return 0;
}

/* Pull (retrive) data from FIFO. Oldest entry from FIFO memory is copied into the provided pDst space. In case of error return value is != 0*/
unsigned long bgFIFOPull(struct bgFIFO_typ* p, unsigned long pDst, unsigned long dstSize)
{
	if(!p)
		return 1;

	if(!p->prvFIFOMemory)
		return 2;

	if(!pDst)
		return 3;

	if(!dstSize || (dstSize != p->cfgEntrySize) )
		return 4;

	if(!p->oFIFOCount)
		return 5;

	p->oPtrPullData = pDst;
	bgFIFOPullEntry(p);
	return 0;
}

/* Get the number of entries stored in the FIFO.*/
unsigned long bgFIFOGetCount(struct bgFIFO_typ* p)
{
	if(!p)
		return 0;

	return p->oFIFOCount;
}

/* Check if FIFO is full.*/
unsigned long bgFIFOIsFull(struct bgFIFO_typ* p)
{
	if(!p)
		return 0;

	return p->oFIFOFull;
}
//EOF
```

#### bgTimer1ms.c
```c
/********************************************************************
 * COPYRIGHT -- pai
 ********************************************************************
 * Package: bglib
 * File: bgTimer1ms.c
 * Author: goran
 * Created: October 05, 2011
 *******************************************************************/
#include <bur/plctypes.h>
#ifdef __cplusplus
	extern "C"
	{
#endif

#include "bglibas.h"

#ifdef __cplusplus
	};
#endif
#include <standard.h>

/* Timer cyclic function. Must be called cyclicly for corret timer operation. */
unsigned long  bgTimerCyclic(struct TON *timer){
	TON(timer);
	return 0;
}

/* Start timer for a defined amount of time [ms]. IMPORTANT: function uses TON library call. Same restrictions apply! */
unsigned long  bgTimerStart(struct TON *timer, unsigned long timeoutTime){
	timer->IN = 0;
	TON(timer);
	timer->IN = 1;
	timer->PT = timeoutTime;
	TON(timer );
	return 0;
}

/* Stop the timer.*/
unsigned long  bgTimerStop(struct TON *timer){
	timer->IN = 0;
	TON(timer);
	return 0;
}

/* Check if timer has expired.*/
BOOL  bgTimerIsTimeOut(struct TON *timer){
	if( bgTimerIsEnabled(timer) ){
		return (timer->Q);
	}else{
		return (1);
	}
}

/* Check if timer is enabled.*/
BOOL  bgTimerIsEnabled(struct TON *timer){
	return (timer->IN);
}

/* Retrive the remainig timer time [ms].*/
unsigned long  bgTimerTimeRemaining(struct TON *timer){
	return (timer->PT - timer->ET);
}

/* Retrive the elapsed timer time [ms].*/
unsigned long  bgTimerTimeElapsed(struct TON *timer) {
	return (timer->ET);
}

//EOF
```

- Program Logical/paiComponents/paiBnRVFD/paiVFDX64 (ANSIC) (no source held here)

### Program Logical/paiComponents/paiFileService
